    # Add subprograms here
    # Start of main program
    # Program generated by RoboDK v5.6.5 for UR10e on 02/02/2024 20:40:15
    # Using nominal kinematics.
    blend_radius_m = 0.001
    speed_ms = 1.000
    # set_reference(p[0.350000, -0.230000, -0.017000, 0.000000, 0.000000, 0.000000])
    set_tcp(p[0.000000, 0.000000, 0.252000, 0.000000, 0.000000, 0.000000])
    # Show Tool
    movej([-0.152532, -1.248081, -2.542110, -0.922198, 1.570796, 1.418264],accel_radss,speed_rads,0,blend_radius_m)
    movel([-0.152532, -1.248081, -2.542110, -0.922198, 1.570796, 1.418264],accel_mss,speed_ms,0,blend_radius_m)
    # Splitting Linear movement in 2 (instruction 7: MoveL 3)
    movel([-0.152532, -1.275419, -2.559682, -0.877288, 1.570796, 1.418264],accel_mss,speed_ms,0,blend_radius_m)
    movel([-0.152532, -1.305068, -2.576535, -0.830786, 1.570796, 1.418264],accel_mss,speed_ms,0,blend_radius_m)
    movel([-0.152532, -1.305068, -2.576535, -0.830786, 1.570796, 1.418264],accel_mss,speed_ms,0,blend_radius_m)
    speed_ms = 1.000
    movel([-0.152532, -1.305068, -2.576535, -0.830786, 1.570796, 1.418264],accel_mss,speed_ms,0,blend_radius_m)
    movel([-0.152532, -1.305068, -2.576535, -0.830786, 1.570796, 1.418264],accel_mss,speed_ms,0,blend_radius_m)
    movel([-0.152532, -1.305068, -2.576535, -0.830786, 1.570796, 1.418264],accel_mss,speed_ms,0,blend_radius_m)
    speed_ms = 0.005
    # Splitting Linear movement in 2 (instruction 14: MoveL 8)
    movel([-0.152532, -1.285041, -2.565382, -0.861966, 1.570796, 1.418264],accel_mss,speed_ms,0,blend_radius_m)
    movel([-0.152532, -1.266054, -2.553902, -0.892433, 1.570796, 1.418264],accel_mss,speed_ms,0,blend_radius_m)
    speed_ms = 1.000
    # Splitting Linear movement in 2 (instruction 16: MoveL 9)
    movel([-0.152532, -1.285041, -2.565382, -0.861966, 1.570796, 1.418264],accel_mss,speed_ms,0,blend_radius_m)
    movel([-0.152532, -1.305068, -2.576535, -0.830786, 1.570796, 1.418264],accel_mss,speed_ms,0,blend_radius_m)
    speed_ms = 0.040
    movel([-0.152532, -1.305068, -2.576535, -0.830786, 1.570796, 1.418264],accel_mss,speed_ms,0,blend_radius_m)
    speed_ms = 1.000
    movel([-0.152532, -1.305068, -2.576535, -0.830786, 1.570796, 1.418264],accel_mss,speed_ms,0,blend_radius_m)
    # Splitting Linear movement in 8 (instruction 21: MoveL 12)
    movel([-0.122948, -1.317915, -2.568481, -0.825992, 1.570796, 1.447849],accel_mss,speed_ms,0,blend_radius_m)
    movel([-0.094642, -1.331738, -2.559579, -0.821073, 1.570796, 1.476154],accel_mss,speed_ms,0,blend_radius_m)
    movel([-0.067601, -1.346424, -2.549844, -0.816120, 1.570796, 1.503196],accel_mss,speed_ms,0,blend_radius_m)
    movel([-0.041798, -1.361869, -2.539298, -0.811223, 1.570796, 1.528999],accel_mss,speed_ms,0,blend_radius_m)
    movel([-0.017201, -1.377969, -2.527959, -0.806462, 1.570796, 1.553595],accel_mss,speed_ms,0,blend_radius_m)
    movel([0.006227, -1.394629, -2.515848, -0.801912, 1.570796, 1.577023],accel_mss,speed_ms,0,blend_radius_m)
    movel([0.028528, -1.411761, -2.502989, -0.797639, 1.570796, 1.599324],accel_mss,speed_ms,0,blend_radius_m)
    movel([0.049747, -1.429285, -2.489403, -0.793702, 1.570796, 1.620543],accel_mss,speed_ms,0,blend_radius_m)
    speed_ms = 0.005
    # Splitting Linear movement in 2 (instruction 23: MoveL 13)
    movel([0.049747, -1.448539, -2.498917, -0.764933, 1.570796, 1.620543],accel_mss,speed_ms,0,blend_radius_m)
    movel([0.049747, -1.468584, -2.508071, -0.735733, 1.570796, 1.620543],accel_mss,speed_ms,0,blend_radius_m)
    speed_ms = 0.025
    movel([0.047987, -1.472694, -2.504618, -0.735077, 1.570796, 1.618783],accel_mss,speed_ms,0,blend_radius_m)
    movel([0.046994, -1.474744, -2.502886, -0.734759, 1.570796, 1.617791],accel_mss,speed_ms,0,blend_radius_m)
    movel([0.045905, -1.476777, -2.501162, -0.734450, 1.570796, 1.616702],accel_mss,speed_ms,0,blend_radius_m)
    movel([0.044706, -1.478782, -2.499455, -0.734152, 1.570796, 1.615502],accel_mss,speed_ms,0,blend_radius_m)
    movel([0.043381, -1.480749, -2.497774, -0.733866, 1.570796, 1.614178],accel_mss,speed_ms,0,blend_radius_m)
    movel([0.041915, -1.482668, -2.496128, -0.733593, 1.570796, 1.612712],accel_mss,speed_ms,0,blend_radius_m)
    movel([0.040291, -1.484527, -2.494529, -0.733333, 1.570796, 1.611088],accel_mss,speed_ms,0,blend_radius_m)
    movel([0.040888, -1.483683, -2.495255, -0.733450, 1.570796, 1.611684],accel_mss,speed_ms,0,blend_radius_m)
    movel([0.041419, -1.482572, -2.496211, -0.733606, 1.570796, 1.612216],accel_mss,speed_ms,0,blend_radius_m)
    movel([0.041720, -1.481480, -2.497148, -0.733761, 1.570796, 1.612517],accel_mss,speed_ms,0,blend_radius_m)
    movel([0.041730, -1.481035, -2.497529, -0.733825, 1.570796, 1.612526],accel_mss,speed_ms,0,blend_radius_m)
    movel([0.041619, -1.480703, -2.497813, -0.733873, 1.570796, 1.612415],accel_mss,speed_ms,0,blend_radius_m)
    movel([0.041364, -1.480515, -2.497974, -0.733900, 1.570796, 1.612160],accel_mss,speed_ms,0,blend_radius_m)
    movel([0.041013, -1.480523, -2.497967, -0.733899, 1.570796, 1.611810],accel_mss,speed_ms,0,blend_radius_m)
    movel([0.040586, -1.480703, -2.497813, -0.733873, 1.570796, 1.611382],accel_mss,speed_ms,0,blend_radius_m)
    movel([0.040090, -1.481034, -2.497530, -0.733825, 1.570796, 1.610886],accel_mss,speed_ms,0,blend_radius_m)
    movel([0.038959, -1.482046, -2.496663, -0.733681, 1.570796, 1.609755],accel_mss,speed_ms,0,blend_radius_m)
    movel([0.037732, -1.483368, -2.495527, -0.733494, 1.570796, 1.608528],accel_mss,speed_ms,0,blend_radius_m)
    movel([0.035425, -1.486199, -2.493085, -0.733105, 1.570796, 1.606222],accel_mss,speed_ms,0,blend_radius_m)
    movel([0.034030, -1.488028, -2.491501, -0.732860, 1.570796, 1.604827],accel_mss,speed_ms,0,blend_radius_m)
    movel([0.031932, -1.490562, -2.489297, -0.732529, 1.570796, 1.602728],accel_mss,speed_ms,0,blend_radius_m)
    movel([0.030757, -1.491738, -2.488272, -0.732379, 1.570796, 1.601553],accel_mss,speed_ms,0,blend_radius_m)
    movel([0.029446, -1.492789, -2.487353, -0.732247, 1.570796, 1.600242],accel_mss,speed_ms,0,blend_radius_m)
    movel([0.029713, -1.492441, -2.487658, -0.732291, 1.570796, 1.600509],accel_mss,speed_ms,0,blend_radius_m)
    movel([0.029890, -1.491885, -2.488143, -0.732361, 1.570796, 1.600686],accel_mss,speed_ms,0,blend_radius_m)
    movel([0.030008, -1.490434, -2.489409, -0.732546, 1.570796, 1.600805],accel_mss,speed_ms,0,blend_radius_m)
    movel([0.029868, -1.489016, -2.490643, -0.732730, 1.570796, 1.600664],accel_mss,speed_ms,0,blend_radius_m)
    movel([0.029718, -1.488499, -2.491093, -0.732798, 1.570796, 1.600514],accel_mss,speed_ms,0,blend_radius_m)
    movel([0.029529, -1.488209, -2.491344, -0.732836, 1.570796, 1.600325],accel_mss,speed_ms,0,blend_radius_m)
    movel([0.028992, -1.487953, -2.491566, -0.732870, 1.570796, 1.599789],accel_mss,speed_ms,0,blend_radius_m)
    movel([0.028458, -1.487944, -2.491574, -0.732871, 1.570796, 1.599254],accel_mss,speed_ms,0,blend_radius_m)
    movel([0.027927, -1.488133, -2.491410, -0.732846, 1.570796, 1.598724],accel_mss,speed_ms,0,blend_radius_m)
    movel([0.027405, -1.488475, -2.491113, -0.732801, 1.570796, 1.598201],accel_mss,speed_ms,0,blend_radius_m)
    movel([0.026411, -1.489409, -2.490302, -0.732678, 1.570796, 1.597207],accel_mss,speed_ms,0,blend_radius_m)
    movel([0.025512, -1.490359, -2.489474, -0.732555, 1.570796, 1.596308],accel_mss,speed_ms,0,blend_radius_m)
    movel([0.024026, -1.491761, -2.488251, -0.732376, 1.570796, 1.594822],accel_mss,speed_ms,0,blend_radius_m)
    movel([0.022503, -1.493004, -2.487165, -0.732220, 1.570796, 1.593300],accel_mss,speed_ms,0,blend_radius_m)
    movel([0.020851, -1.494060, -2.486240, -0.732089, 1.570796, 1.591648],accel_mss,speed_ms,0,blend_radius_m)
    movel([0.018986, -1.494894, -2.485508, -0.731987, 1.570796, 1.589782],accel_mss,speed_ms,0,blend_radius_m)
    movel([0.020018, -1.493786, -2.486480, -0.732123, 1.570796, 1.590814],accel_mss,speed_ms,0,blend_radius_m)
    movel([0.020844, -1.492612, -2.487508, -0.732269, 1.570796, 1.591641],accel_mss,speed_ms,0,blend_radius_m)
    movel([0.021097, -1.491990, -2.488052, -0.732347, 1.570796, 1.591893],accel_mss,speed_ms,0,blend_radius_m)
    movel([0.021184, -1.491389, -2.488577, -0.732423, 1.570796, 1.591981],accel_mss,speed_ms,0,blend_radius_m)
    movel([0.021086, -1.490859, -2.489039, -0.732491, 1.570796, 1.591883],accel_mss,speed_ms,0,blend_radius_m)
    movel([0.020770, -1.490458, -2.489389, -0.732543, 1.570796, 1.591566],accel_mss,speed_ms,0,blend_radius_m)
    movel([0.020101, -1.490219, -2.489596, -0.732573, 1.570796, 1.590897],accel_mss,speed_ms,0,blend_radius_m)
    movel([0.019264, -1.490254, -2.489566, -0.732569, 1.570796, 1.590061],accel_mss,speed_ms,0,blend_radius_m)
    movel([0.018340, -1.490477, -2.489372, -0.732540, 1.570796, 1.589137],accel_mss,speed_ms,0,blend_radius_m)
    movel([0.017414, -1.490797, -2.489093, -0.732499, 1.570796, 1.588211],accel_mss,speed_ms,0,blend_radius_m)
    speed_ms = 0.005
    movel([0.017414, -1.482861, -2.485566, -0.743963, 1.570796, 1.588211],accel_mss,speed_ms,0,blend_radius_m)
    speed_ms = 0.040
    movel([0.019926, -1.498929, -2.471530, -0.741930, 1.570796, 1.590722],accel_mss,speed_ms,0,blend_radius_m)
    speed_ms = 0.005
    movel([0.019926, -1.506737, -2.474994, -0.730658, 1.570796, 1.590722],accel_mss,speed_ms,0,blend_radius_m)
    speed_ms = 0.025
    movel([0.020345, -1.505703, -2.475921, -0.730765, 1.570796, 1.591141],accel_mss,speed_ms,0,blend_radius_m)
    movel([0.020900, -1.504675, -2.476841, -0.730873, 1.570796, 1.591696],accel_mss,speed_ms,0,blend_radius_m)
    movel([0.021577, -1.503669, -2.477739, -0.730981, 1.570796, 1.592373],accel_mss,speed_ms,0,blend_radius_m)
    movel([0.022366, -1.502696, -2.478607, -0.731086, 1.570796, 1.593163],accel_mss,speed_ms,0,blend_radius_m)
    movel([0.023256, -1.501770, -2.479431, -0.731188, 1.570796, 1.594052],accel_mss,speed_ms,0,blend_radius_m)
    movel([0.024233, -1.500906, -2.480198, -0.731285, 1.570796, 1.595030],accel_mss,speed_ms,0,blend_radius_m)
    movel([0.025286, -1.500119, -2.480897, -0.731373, 1.570796, 1.596082],accel_mss,speed_ms,0,blend_radius_m)
    movel([0.026405, -1.499419, -2.481517, -0.731453, 1.570796, 1.597201],accel_mss,speed_ms,0,blend_radius_m)
    movel([0.028138, -1.498558, -2.482279, -0.731552, 1.570796, 1.598935],accel_mss,speed_ms,0,blend_radius_m)
    movel([0.029837, -1.497950, -2.482816, -0.731623, 1.570796, 1.600634],accel_mss,speed_ms,0,blend_radius_m)
    movel([0.031496, -1.497576, -2.483146, -0.731667, 1.570796, 1.602293],accel_mss,speed_ms,0,blend_radius_m)
    movel([0.033106, -1.497418, -2.483285, -0.731685, 1.570796, 1.603903],accel_mss,speed_ms,0,blend_radius_m)
    movel([0.034662, -1.497458, -2.483250, -0.731681, 1.570796, 1.605458],accel_mss,speed_ms,0,blend_radius_m)
    movel([0.036159, -1.497677, -2.483057, -0.731655, 1.570796, 1.606956],accel_mss,speed_ms,0,blend_radius_m)
    movel([0.037589, -1.498057, -2.482722, -0.731610, 1.570796, 1.608386],accel_mss,speed_ms,0,blend_radius_m)
    movel([0.038948, -1.498578, -2.482261, -0.731550, 1.570796, 1.609744],accel_mss,speed_ms,0,blend_radius_m)
    movel([0.040230, -1.499221, -2.481692, -0.731476, 1.570796, 1.611026],accel_mss,speed_ms,0,blend_radius_m)
    movel([0.041430, -1.499967, -2.481031, -0.731391, 1.570796, 1.612227],accel_mss,speed_ms,0,blend_radius_m)
    movel([0.043569, -1.501692, -2.479500, -0.731197, 1.570796, 1.614365],accel_mss,speed_ms,0,blend_radius_m)
    movel([0.045328, -1.503594, -2.477806, -0.730989, 1.570796, 1.616124],accel_mss,speed_ms,0,blend_radius_m)
    movel([0.046669, -1.505525, -2.476080, -0.730784, 1.570796, 1.617465],accel_mss,speed_ms,0,blend_radius_m)
    movel([0.047792, -1.507678, -2.474150, -0.730562, 1.570796, 1.618588],accel_mss,speed_ms,0,blend_radius_m)
    movel([0.048705, -1.509943, -2.472110, -0.730336, 1.570796, 1.619501],accel_mss,speed_ms,0,blend_radius_m)
    movel([0.049431, -1.512301, -2.469978, -0.730110, 1.570796, 1.620227],accel_mss,speed_ms,0,blend_radius_m)
    movel([0.049991, -1.514735, -2.467768, -0.729886, 1.570796, 1.620788],accel_mss,speed_ms,0,blend_radius_m)
    movel([0.050411, -1.517225, -2.465497, -0.729667, 1.570796, 1.621207],accel_mss,speed_ms,0,blend_radius_m)
    movel([0.050713, -1.519754, -2.463181, -0.729454, 1.570796, 1.621510],accel_mss,speed_ms,0,blend_radius_m)
    movel([0.051058, -1.524854, -2.458479, -0.729056, 1.570796, 1.621854],accel_mss,speed_ms,0,blend_radius_m)
    movel([0.051259, -1.528417, -2.455169, -0.728803, 1.570796, 1.622055],accel_mss,speed_ms,0,blend_radius_m)
    movel([0.051521, -1.530125, -2.453575, -0.728689, 1.570796, 1.622318],accel_mss,speed_ms,0,blend_radius_m)
    movel([0.051999, -1.531735, -2.452069, -0.728586, 1.570796, 1.622795],accel_mss,speed_ms,0,blend_radius_m)
    movel([0.052951, -1.533693, -2.450230, -0.728465, 1.570796, 1.623747],accel_mss,speed_ms,0,blend_radius_m)
    movel([0.053905, -1.535658, -2.448380, -0.728351, 1.570796, 1.624701],accel_mss,speed_ms,0,blend_radius_m)
    movel([0.054234, -1.536676, -2.447418, -0.728294, 1.570796, 1.625030],accel_mss,speed_ms,0,blend_radius_m)
    movel([0.054384, -1.537737, -2.446415, -0.728237, 1.570796, 1.625180],accel_mss,speed_ms,0,blend_radius_m)
    movel([0.054296, -1.538850, -2.445360, -0.728179, 1.570796, 1.625093],accel_mss,speed_ms,0,blend_radius_m)
    movel([0.053915, -1.540032, -2.444238, -0.728119, 1.570796, 1.624711],accel_mss,speed_ms,0,blend_radius_m)
    movel([0.055176, -1.537118, -2.447000, -0.728270, 1.570796, 1.625972],accel_mss,speed_ms,0,blend_radius_m)
    movel([0.056268, -1.534210, -2.449744, -0.728435, 1.570796, 1.627064],accel_mss,speed_ms,0,blend_radius_m)
    movel([0.058142, -1.528367, -2.455216, -0.728806, 1.570796, 1.628938],accel_mss,speed_ms,0,blend_radius_m)
    movel([0.059066, -1.525102, -2.458249, -0.729038, 1.570796, 1.629862],accel_mss,speed_ms,0,blend_radius_m)
    movel([0.059888, -1.521837, -2.461266, -0.729287, 1.570796, 1.630684],accel_mss,speed_ms,0,blend_radius_m)
    movel([0.061298, -1.515293, -2.467260, -0.729836, 1.570796, 1.632094],accel_mss,speed_ms,0,blend_radius_m)
    movel([0.062426, -1.508876, -2.473071, -0.730441, 1.570796, 1.633222],accel_mss,speed_ms,0,blend_radius_m)
    movel([0.062809, -1.505673, -2.475948, -0.730768, 1.570796, 1.633605],accel_mss,speed_ms,0,blend_radius_m)
    movel([0.062991, -1.502530, -2.478754, -0.731105, 1.570796, 1.633787],accel_mss,speed_ms,0,blend_radius_m)
    movel([0.062929, -1.500110, -2.480905, -0.731374, 1.570796, 1.633725],accel_mss,speed_ms,0,blend_radius_m)
    movel([0.062735, -1.497714, -2.483025, -0.731651, 1.570796, 1.633532],accel_mss,speed_ms,0,blend_radius_m)
    movel([0.062551, -1.495294, -2.485157, -0.731939, 1.570796, 1.633347],accel_mss,speed_ms,0,blend_radius_m)
    movel([0.062514, -1.492802, -2.487341, -0.732245, 1.570796, 1.633310],accel_mss,speed_ms,0,blend_radius_m)
    movel([0.062598, -1.492115, -2.487942, -0.732331, 1.570796, 1.633394],accel_mss,speed_ms,0,blend_radius_m)
    movel([0.062833, -1.491405, -2.488563, -0.732421, 1.570796, 1.633629],accel_mss,speed_ms,0,blend_radius_m)
    movel([0.063253, -1.490783, -2.489105, -0.732501, 1.570796, 1.634049],accel_mss,speed_ms,0,blend_radius_m)
    movel([0.063548, -1.490538, -2.489318, -0.732532, 1.570796, 1.634344],accel_mss,speed_ms,0,blend_radius_m)
    movel([0.063906, -1.490355, -2.489478, -0.732556, 1.570796, 1.634702],accel_mss,speed_ms,0,blend_radius_m)
    movel([0.064424, -1.490247, -2.489573, -0.732570, 1.570796, 1.635220],accel_mss,speed_ms,0,blend_radius_m)
    movel([0.064916, -1.490252, -2.489568, -0.732569, 1.570796, 1.635712],accel_mss,speed_ms,0,blend_radius_m)
    movel([0.067510, -1.490558, -2.489301, -0.732530, 1.570796, 1.638306],accel_mss,speed_ms,0,blend_radius_m)
    movel([0.069847, -1.491127, -2.488805, -0.732457, 1.570796, 1.640644],accel_mss,speed_ms,0,blend_radius_m)
    movel([0.071947, -1.491931, -2.488103, -0.732355, 1.570796, 1.642743],accel_mss,speed_ms,0,blend_radius_m)
    movel([0.073826, -1.492954, -2.487208, -0.732226, 1.570796, 1.644622],accel_mss,speed_ms,0,blend_radius_m)
    movel([0.075502, -1.494170, -2.486143, -0.732076, 1.570796, 1.646298],accel_mss,speed_ms,0,blend_radius_m)
    movel([0.076994, -1.495556, -2.484926, -0.731907, 1.570796, 1.647790],accel_mss,speed_ms,0,blend_radius_m)
    movel([0.078319, -1.497090, -2.483575, -0.731724, 1.570796, 1.649115],accel_mss,speed_ms,0,blend_radius_m)
    movel([0.079494, -1.498753, -2.482106, -0.731530, 1.570796, 1.650290],accel_mss,speed_ms,0,blend_radius_m)
    movel([0.080539, -1.500520, -2.480541, -0.731328, 1.570796, 1.651335],accel_mss,speed_ms,0,blend_radius_m)
    movel([0.081473, -1.502370, -2.478897, -0.731122, 1.570796, 1.652270],accel_mss,speed_ms,0,blend_radius_m)
    movel([0.083080, -1.506232, -2.475447, -0.730710, 1.570796, 1.653876],accel_mss,speed_ms,0,blend_radius_m)
    movel([0.085758, -1.514035, -2.468404, -0.729950, 1.570796, 1.656554],accel_mss,speed_ms,0,blend_radius_m)
    movel([0.086253, -1.515217, -2.467329, -0.729843, 1.570796, 1.657050],accel_mss,speed_ms,0,blend_radius_m)
    movel([0.086622, -1.515721, -2.466870, -0.729798, 1.570796, 1.657418],accel_mss,speed_ms,0,blend_radius_m)
    movel([0.087122, -1.516115, -2.466511, -0.729763, 1.570796, 1.657919],accel_mss,speed_ms,0,blend_radius_m)
    movel([0.088103, -1.516424, -2.466228, -0.729736, 1.570796, 1.658899],accel_mss,speed_ms,0,blend_radius_m)
    movel([0.088627, -1.516441, -2.466213, -0.729735, 1.570796, 1.659423],accel_mss,speed_ms,0,blend_radius_m)
    movel([0.089168, -1.516374, -2.466274, -0.729741, 1.570796, 1.659965],accel_mss,speed_ms,0,blend_radius_m)
    movel([0.090276, -1.516027, -2.466591, -0.729771, 1.570796, 1.661072],accel_mss,speed_ms,0,blend_radius_m)
    movel([0.091387, -1.515445, -2.467122, -0.729823, 1.570796, 1.662183],accel_mss,speed_ms,0,blend_radius_m)
    movel([0.092457, -1.514694, -2.467805, -0.729890, 1.570796, 1.663254],accel_mss,speed_ms,0,blend_radius_m)
    movel([0.093445, -1.513838, -2.468584, -0.729968, 1.570796, 1.664242],accel_mss,speed_ms,0,blend_radius_m)
    movel([0.094311, -1.512937, -2.469401, -0.730051, 1.570796, 1.665107],accel_mss,speed_ms,0,blend_radius_m)
    movel([0.095004, -1.512057, -2.470199, -0.730133, 1.570796, 1.665800],accel_mss,speed_ms,0,blend_radius_m)
    movel([0.096042, -1.510510, -2.471598, -0.730281, 1.570796, 1.666838],accel_mss,speed_ms,0,blend_radius_m)
    movel([0.097003, -1.508932, -2.473021, -0.730436, 1.570796, 1.667799],accel_mss,speed_ms,0,blend_radius_m)
    movel([0.098688, -1.505713, -2.475912, -0.730764, 1.570796, 1.669484],accel_mss,speed_ms,0,blend_radius_m)
    movel([0.100061, -1.502456, -2.478820, -0.731113, 1.570796, 1.670857],accel_mss,speed_ms,0,blend_radius_m)
    movel([0.101119, -1.499219, -2.481694, -0.731476, 1.570796, 1.671915],accel_mss,speed_ms,0,blend_radius_m)
    movel([0.101462, -1.498003, -2.482769, -0.731617, 1.570796, 1.672258],accel_mss,speed_ms,0,blend_radius_m)
    movel([0.101921, -1.496793, -2.483837, -0.731759, 1.570796, 1.672717],accel_mss,speed_ms,0,blend_radius_m)
    movel([0.102246, -1.496209, -2.484351, -0.731829, 1.570796, 1.673043],accel_mss,speed_ms,0,blend_radius_m)
    movel([0.102663, -1.495646, -2.484847, -0.731896, 1.570796, 1.673459],accel_mss,speed_ms,0,blend_radius_m)
    movel([0.103191, -1.495113, -2.485315, -0.731961, 1.570796, 1.673987],accel_mss,speed_ms,0,blend_radius_m)
    movel([0.103850, -1.494618, -2.485750, -0.732021, 1.570796, 1.674647],accel_mss,speed_ms,0,blend_radius_m)
    movel([0.104844, -1.494159, -2.486153, -0.732077, 1.570796, 1.675640],accel_mss,speed_ms,0,blend_radius_m)
    movel([0.105852, -1.494002, -2.486291, -0.732096, 1.570796, 1.676648],accel_mss,speed_ms,0,blend_radius_m)
    movel([0.106800, -1.494096, -2.486208, -0.732085, 1.570796, 1.677597],accel_mss,speed_ms,0,blend_radius_m)
    movel([0.107623, -1.494391, -2.485949, -0.732049, 1.570796, 1.678419],accel_mss,speed_ms,0,blend_radius_m)
    movel([0.108793, -1.495109, -2.485319, -0.731961, 1.570796, 1.679590],accel_mss,speed_ms,0,blend_radius_m)
    movel([0.109841, -1.495969, -2.484562, -0.731857, 1.570796, 1.680638],accel_mss,speed_ms,0,blend_radius_m)
    movel([0.111647, -1.497907, -2.482854, -0.731628, 1.570796, 1.682444],accel_mss,speed_ms,0,blend_radius_m)
    movel([0.112379, -1.498899, -2.481977, -0.731513, 1.570796, 1.683175],accel_mss,speed_ms,0,blend_radius_m)
    movel([0.112973, -1.499942, -2.481054, -0.731393, 1.570796, 1.683770],accel_mss,speed_ms,0,blend_radius_m)
    movel([0.113440, -1.501029, -2.480089, -0.731271, 1.570796, 1.684237],accel_mss,speed_ms,0,blend_radius_m)
    movel([0.113785, -1.502160, -2.479084, -0.731145, 1.570796, 1.684581],accel_mss,speed_ms,0,blend_radius_m)
    movel([0.114013, -1.503328, -2.478044, -0.731018, 1.570796, 1.684810],accel_mss,speed_ms,0,blend_radius_m)
    movel([0.114151, -1.505768, -2.475863, -0.730758, 1.570796, 1.684947],accel_mss,speed_ms,0,blend_radius_m)
    movel([0.114072, -1.507032, -2.474729, -0.730628, 1.570796, 1.684869],accel_mss,speed_ms,0,blend_radius_m)
    movel([0.113660, -1.509630, -2.472392, -0.730367, 1.570796, 1.684456],accel_mss,speed_ms,0,blend_radius_m)
    movel([0.112946, -1.512298, -2.469980, -0.730110, 1.570796, 1.683743],accel_mss,speed_ms,0,blend_radius_m)
    movel([0.111984, -1.515015, -2.467513, -0.729861, 1.570796, 1.682780],accel_mss,speed_ms,0,blend_radius_m)
    movel([0.110827, -1.517747, -2.465020, -0.729622, 1.570796, 1.681624],accel_mss,speed_ms,0,blend_radius_m)
    movel([0.108876, -1.521723, -2.461371, -0.729296, 1.570796, 1.679673],accel_mss,speed_ms,0,blend_radius_m)
    movel([0.107771, -1.523695, -2.459551, -0.729143, 1.570796, 1.678567],accel_mss,speed_ms,0,blend_radius_m)
    movel([0.106563, -1.525642, -2.457749, -0.728999, 1.570796, 1.677359],accel_mss,speed_ms,0,blend_radius_m)
    movel([0.105242, -1.527548, -2.455978, -0.728863, 1.570796, 1.676038],accel_mss,speed_ms,0,blend_radius_m)
    movel([0.103799, -1.529403, -2.454250, -0.728737, 1.570796, 1.674595],accel_mss,speed_ms,0,blend_radius_m)
    movel([0.102219, -1.531196, -2.452573, -0.728620, 1.570796, 1.673015],accel_mss,speed_ms,0,blend_radius_m)
    movel([0.100495, -1.532914, -2.450963, -0.728513, 1.570796, 1.671291],accel_mss,speed_ms,0,blend_radius_m)
    movel([0.097886, -1.535185, -2.448826, -0.728378, 1.570796, 1.668682],accel_mss,speed_ms,0,blend_radius_m)
    movel([0.096431, -1.536300, -2.447774, -0.728315, 1.570796, 1.667227],accel_mss,speed_ms,0,blend_radius_m)
    movel([0.094906, -1.537331, -2.446799, -0.728259, 1.570796, 1.665702],accel_mss,speed_ms,0,blend_radius_m)
    movel([0.093336, -1.538226, -2.445951, -0.728211, 1.570796, 1.664133],accel_mss,speed_ms,0,blend_radius_m)
    movel([0.091746, -1.538933, -2.445281, -0.728174, 1.570796, 1.662542],accel_mss,speed_ms,0,blend_radius_m)
    movel([0.090156, -1.539398, -2.444841, -0.728151, 1.570796, 1.660953],accel_mss,speed_ms,0,blend_radius_m)
    movel([0.089370, -1.539524, -2.444720, -0.728144, 1.570796, 1.660167],accel_mss,speed_ms,0,blend_radius_m)
    movel([0.088595, -1.539569, -2.444678, -0.728142, 1.570796, 1.659391],accel_mss,speed_ms,0,blend_radius_m)
    movel([0.087751, -1.539517, -2.444727, -0.728145, 1.570796, 1.658547],accel_mss,speed_ms,0,blend_radius_m)
    movel([0.086976, -1.539361, -2.444875, -0.728153, 1.570796, 1.657772],accel_mss,speed_ms,0,blend_radius_m)
    movel([0.086265, -1.539111, -2.445113, -0.728165, 1.570796, 1.657062],accel_mss,speed_ms,0,blend_radius_m)
    movel([0.085615, -1.538774, -2.445432, -0.728183, 1.570796, 1.656412],accel_mss,speed_ms,0,blend_radius_m)
    movel([0.084479, -1.537886, -2.446274, -0.728229, 1.570796, 1.655275],accel_mss,speed_ms,0,blend_radius_m)
    movel([0.083539, -1.536771, -2.447329, -0.728289, 1.570796, 1.654335],accel_mss,speed_ms,0,blend_radius_m)
    movel([0.082764, -1.535510, -2.448519, -0.728360, 1.570796, 1.653560],accel_mss,speed_ms,0,blend_radius_m)
    movel([0.082122, -1.534181, -2.449771, -0.728436, 1.570796, 1.652919],accel_mss,speed_ms,0,blend_radius_m)
    movel([0.081123, -1.531634, -2.452163, -0.728592, 1.570796, 1.651920],accel_mss,speed_ms,0,blend_radius_m)
    movel([0.080674, -1.530439, -2.453281, -0.728668, 1.570796, 1.651470],accel_mss,speed_ms,0,blend_radius_m)
    movel([0.080087, -1.529336, -2.454312, -0.728741, 1.570796, 1.650883],accel_mss,speed_ms,0,blend_radius_m)
    movel([0.079683, -1.528878, -2.454739, -0.728772, 1.570796, 1.650479],accel_mss,speed_ms,0,blend_radius_m)
    movel([0.079173, -1.528514, -2.455079, -0.728796, 1.570796, 1.649970],accel_mss,speed_ms,0,blend_radius_m)
    movel([0.078537, -1.528269, -2.455307, -0.728813, 1.570796, 1.649333],accel_mss,speed_ms,0,blend_radius_m)
    movel([0.077749, -1.528165, -2.455404, -0.728820, 1.570796, 1.648545],accel_mss,speed_ms,0,blend_radius_m)
    movel([0.077921, -1.528219, -2.455353, -0.728817, 1.570796, 1.648717],accel_mss,speed_ms,0,blend_radius_m)
    movel([0.078022, -1.528366, -2.455217, -0.728807, 1.570796, 1.648818],accel_mss,speed_ms,0,blend_radius_m)
    movel([0.078024, -1.528912, -2.454707, -0.728769, 1.570796, 1.648821],accel_mss,speed_ms,0,blend_radius_m)
    movel([0.077786, -1.529757, -2.453919, -0.728713, 1.570796, 1.648582],accel_mss,speed_ms,0,blend_radius_m)
    movel([0.077343, -1.530853, -2.452894, -0.728642, 1.570796, 1.648140],accel_mss,speed_ms,0,blend_radius_m)
    movel([0.075981, -1.533606, -2.450312, -0.728471, 1.570796, 1.646777],accel_mss,speed_ms,0,blend_radius_m)
    movel([0.074205, -1.536791, -2.447310, -0.728288, 1.570796, 1.645001],accel_mss,speed_ms,0,blend_radius_m)
    movel([0.070469, -1.542969, -2.441439, -0.727980, 1.570796, 1.641265],accel_mss,speed_ms,0,blend_radius_m)
    movel([0.068192, -1.546458, -2.438097, -0.727834, 1.570796, 1.638988],accel_mss,speed_ms,0,blend_radius_m)
    movel([0.065488, -1.549998, -2.434686, -0.727705, 1.570796, 1.636284],accel_mss,speed_ms,0,blend_radius_m)
    movel([0.062729, -1.553454, -2.431336, -0.727599, 1.570796, 1.633525],accel_mss,speed_ms,0,blend_radius_m)
    movel([0.059905, -1.556864, -2.428013, -0.727513, 1.570796, 1.630702],accel_mss,speed_ms,0,blend_radius_m)
    movel([0.054252, -1.563384, -2.421604, -0.727401, 1.570796, 1.625048],accel_mss,speed_ms,0,blend_radius_m)
    movel([0.051363, -1.566407, -2.418610, -0.727372, 1.570796, 1.622159],accel_mss,speed_ms,0,blend_radius_m)
    movel([0.049836, -1.567837, -2.417189, -0.727363, 1.570796, 1.620632],accel_mss,speed_ms,0,blend_radius_m)
    movel([0.048242, -1.569190, -2.415840, -0.727358, 1.570796, 1.619039],accel_mss,speed_ms,0,blend_radius_m)
    movel([0.046566, -1.570450, -2.414583, -0.727356, 1.570796, 1.617363],accel_mss,speed_ms,0,blend_radius_m)
    movel([0.044802, -1.571600, -2.413433, -0.727357, 1.570796, 1.615598],accel_mss,speed_ms,0,blend_radius_m)
    movel([0.045149, -1.568689, -2.416340, -0.727360, 1.570796, 1.615946],accel_mss,speed_ms,0,blend_radius_m)
    movel([0.045119, -1.567858, -2.417168, -0.727363, 1.570796, 1.615916],accel_mss,speed_ms,0,blend_radius_m)
    movel([0.044947, -1.567542, -2.417483, -0.727365, 1.570796, 1.615743],accel_mss,speed_ms,0,blend_radius_m)
    movel([0.044607, -1.567377, -2.417647, -0.727366, 1.570796, 1.615403],accel_mss,speed_ms,0,blend_radius_m)
    movel([0.044234, -1.567394, -2.417629, -0.727366, 1.570796, 1.615030],accel_mss,speed_ms,0,blend_radius_m)
    movel([0.043838, -1.567527, -2.417497, -0.727365, 1.570796, 1.614635],accel_mss,speed_ms,0,blend_radius_m)
    movel([0.041962, -1.568497, -2.416532, -0.727361, 1.570796, 1.612759],accel_mss,speed_ms,0,blend_radius_m)
    movel([0.040849, -1.568905, -2.416124, -0.727359, 1.570796, 1.611646],accel_mss,speed_ms,0,blend_radius_m)
    movel([0.039732, -1.569172, -2.415858, -0.727358, 1.570796, 1.610528],accel_mss,speed_ms,0,blend_radius_m)
    movel([0.038640, -1.569290, -2.415741, -0.727358, 1.570796, 1.609436],accel_mss,speed_ms,0,blend_radius_m)
    movel([0.038311, -1.569242, -2.415789, -0.727358, 1.570796, 1.609108],accel_mss,speed_ms,0,blend_radius_m)
    movel([0.038215, -1.569055, -2.415975, -0.727359, 1.570796, 1.609011],accel_mss,speed_ms,0,blend_radius_m)
    movel([0.038508, -1.568213, -2.416814, -0.727362, 1.570796, 1.609304],accel_mss,speed_ms,0,blend_radius_m)
    movel([0.038473, -1.567947, -2.417080, -0.727363, 1.570796, 1.609269],accel_mss,speed_ms,0,blend_radius_m)
    movel([0.038291, -1.567758, -2.417267, -0.727364, 1.570796, 1.609087],accel_mss,speed_ms,0,blend_radius_m)
    movel([0.038010, -1.567656, -2.417369, -0.727364, 1.570796, 1.608806],accel_mss,speed_ms,0,blend_radius_m)
    movel([0.037675, -1.567648, -2.417377, -0.727364, 1.570796, 1.608472],accel_mss,speed_ms,0,blend_radius_m)
    movel([0.036971, -1.567857, -2.417169, -0.727363, 1.570796, 1.607768],accel_mss,speed_ms,0,blend_radius_m)
    movel([0.032034, -1.570539, -2.414494, -0.727356, 1.570796, 1.602831],accel_mss,speed_ms,0,blend_radius_m)
    movel([0.033488, -1.569504, -2.415528, -0.727358, 1.570796, 1.604284],accel_mss,speed_ms,0,blend_radius_m)
    movel([0.034915, -1.568368, -2.416660, -0.727361, 1.570796, 1.605712],accel_mss,speed_ms,0,blend_radius_m)
    movel([0.036304, -1.567153, -2.417869, -0.727367, 1.570796, 1.607100],accel_mss,speed_ms,0,blend_radius_m)
    movel([0.037649, -1.565876, -2.419138, -0.727376, 1.570796, 1.608445],accel_mss,speed_ms,0,blend_radius_m)
    movel([0.040174, -1.563204, -2.421782, -0.727403, 1.570796, 1.610970],accel_mss,speed_ms,0,blend_radius_m)
    movel([0.042420, -1.560504, -2.424443, -0.727442, 1.570796, 1.613216],accel_mss,speed_ms,0,blend_radius_m)
    movel([0.044692, -1.557524, -2.427367, -0.727498, 1.570796, 1.615489],accel_mss,speed_ms,0,blend_radius_m)
    movel([0.046838, -1.554469, -2.430349, -0.727571, 1.570796, 1.617635],accel_mss,speed_ms,0,blend_radius_m)
    movel([0.047827, -1.552916, -2.431859, -0.727614, 1.570796, 1.618623],accel_mss,speed_ms,0,blend_radius_m)
    movel([0.048742, -1.551347, -2.433381, -0.727661, 1.570796, 1.619539],accel_mss,speed_ms,0,blend_radius_m)
    movel([0.049567, -1.549765, -2.434911, -0.727713, 1.570796, 1.620363],accel_mss,speed_ms,0,blend_radius_m)
    movel([0.050288, -1.548168, -2.436452, -0.727769, 1.570796, 1.621084],accel_mss,speed_ms,0,blend_radius_m)
    movel([0.050654, -1.547170, -2.437413, -0.727806, 1.570796, 1.621451],accel_mss,speed_ms,0,blend_radius_m)
    movel([0.050929, -1.546167, -2.438377, -0.727845, 1.570796, 1.621725],accel_mss,speed_ms,0,blend_radius_m)
    movel([0.051225, -1.544162, -2.440299, -0.727928, 1.570796, 1.622021],accel_mss,speed_ms,0,blend_radius_m)
    movel([0.051211, -1.542184, -2.442189, -0.728016, 1.570796, 1.622007],accel_mss,speed_ms,0,blend_radius_m)
    movel([0.050919, -1.540264, -2.444018, -0.728108, 1.570796, 1.621716],accel_mss,speed_ms,0,blend_radius_m)
    movel([0.050389, -1.538428, -2.445760, -0.728201, 1.570796, 1.621186],accel_mss,speed_ms,0,blend_radius_m)
    movel([0.049659, -1.536708, -2.447388, -0.728293, 1.570796, 1.620455],accel_mss,speed_ms,0,blend_radius_m)
    movel([0.048760, -1.535134, -2.448874, -0.728381, 1.570796, 1.619557],accel_mss,speed_ms,0,blend_radius_m)
    movel([0.047734, -1.533734, -2.450192, -0.728463, 1.570796, 1.618531],accel_mss,speed_ms,0,blend_radius_m)
    movel([0.046969, -1.533087, -2.450800, -0.728502, 1.570796, 1.617766],accel_mss,speed_ms,0,blend_radius_m)
    movel([0.046036, -1.532733, -2.451133, -0.728524, 1.570796, 1.616832],accel_mss,speed_ms,0,blend_radius_m)
    movel([0.044989, -1.532658, -2.451202, -0.728528, 1.570796, 1.615785],accel_mss,speed_ms,0,blend_radius_m)
    movel([0.043886, -1.532851, -2.451022, -0.728516, 1.570796, 1.614683],accel_mss,speed_ms,0,blend_radius_m)
    movel([0.042779, -1.533292, -2.450607, -0.728490, 1.570796, 1.613575],accel_mss,speed_ms,0,blend_radius_m)
    movel([0.041722, -1.533971, -2.449969, -0.728449, 1.570796, 1.612519],accel_mss,speed_ms,0,blend_radius_m)
    movel([0.040776, -1.534867, -2.449125, -0.728396, 1.570796, 1.611572],accel_mss,speed_ms,0,blend_radius_m)
    movel([0.039990, -1.535966, -2.448089, -0.728334, 1.570796, 1.610787],accel_mss,speed_ms,0,blend_radius_m)
    movel([0.038953, -1.537691, -2.446459, -0.728239, 1.570796, 1.609749],accel_mss,speed_ms,0,blend_radius_m)
    movel([0.037826, -1.539382, -2.444855, -0.728152, 1.570796, 1.608622],accel_mss,speed_ms,0,blend_radius_m)
    movel([0.036599, -1.541021, -2.443297, -0.728071, 1.570796, 1.607395],accel_mss,speed_ms,0,blend_radius_m)
    movel([0.035257, -1.542593, -2.441799, -0.727997, 1.570796, 1.606053],accel_mss,speed_ms,0,blend_radius_m)
    movel([0.033791, -1.544077, -2.440380, -0.727932, 1.570796, 1.604587],accel_mss,speed_ms,0,blend_radius_m)
    movel([0.032187, -1.545460, -2.439055, -0.727874, 1.570796, 1.602984],accel_mss,speed_ms,0,blend_radius_m)
    movel([0.030433, -1.546725, -2.437841, -0.727823, 1.570796, 1.601229],accel_mss,speed_ms,0,blend_radius_m)
    movel([0.028519, -1.547854, -2.436755, -0.727781, 1.570796, 1.599315],accel_mss,speed_ms,0,blend_radius_m)
    movel([0.027475, -1.548332, -2.436294, -0.727763, 1.570796, 1.598272],accel_mss,speed_ms,0,blend_radius_m)
    movel([0.026412, -1.548698, -2.435941, -0.727750, 1.570796, 1.597208],accel_mss,speed_ms,0,blend_radius_m)
    movel([0.024268, -1.549225, -2.435433, -0.727731, 1.570796, 1.595065],accel_mss,speed_ms,0,blend_radius_m)
    movel([0.022596, -1.549491, -2.435176, -0.727722, 1.570796, 1.593392],accel_mss,speed_ms,0,blend_radius_m)
    movel([0.021010, -1.549563, -2.435106, -0.727720, 1.570796, 1.591806],accel_mss,speed_ms,0,blend_radius_m)
    movel([0.019511, -1.549457, -2.435209, -0.727723, 1.570796, 1.590308],accel_mss,speed_ms,0,blend_radius_m)
    movel([0.018095, -1.549187, -2.435470, -0.727733, 1.570796, 1.588891],accel_mss,speed_ms,0,blend_radius_m)
    movel([0.016758, -1.548771, -2.435871, -0.727747, 1.570796, 1.587554],accel_mss,speed_ms,0,blend_radius_m)
    movel([0.015496, -1.548222, -2.436399, -0.727767, 1.570796, 1.586293],accel_mss,speed_ms,0,blend_radius_m)
    movel([0.014313, -1.547556, -2.437041, -0.727792, 1.570796, 1.585109],accel_mss,speed_ms,0,blend_radius_m)
    movel([0.013202, -1.546790, -2.437779, -0.727821, 1.570796, 1.583999],accel_mss,speed_ms,0,blend_radius_m)
    movel([0.012162, -1.545938, -2.438597, -0.727854, 1.570796, 1.582959],accel_mss,speed_ms,0,blend_radius_m)
    movel([0.011193, -1.545012, -2.439485, -0.727892, 1.570796, 1.581989],accel_mss,speed_ms,0,blend_radius_m)
    movel([0.009457, -1.543013, -2.441397, -0.727978, 1.570796, 1.580253],accel_mss,speed_ms,0,blend_radius_m)
    movel([0.007979, -1.540912, -2.443401, -0.728076, 1.570796, 1.578775],accel_mss,speed_ms,0,blend_radius_m)
    movel([0.006747, -1.538836, -2.445373, -0.728179, 1.570796, 1.577544],accel_mss,speed_ms,0,blend_radius_m)
    movel([0.005914, -1.537189, -2.446933, -0.728266, 1.570796, 1.576710],accel_mss,speed_ms,0,blend_radius_m)
    movel([0.005168, -1.535434, -2.448591, -0.728364, 1.570796, 1.575964],accel_mss,speed_ms,0,blend_radius_m)
    movel([0.004519, -1.533579, -2.450338, -0.728472, 1.570796, 1.575315],accel_mss,speed_ms,0,blend_radius_m)
    movel([0.003986, -1.531636, -2.452161, -0.728592, 1.570796, 1.574783],accel_mss,speed_ms,0,blend_radius_m)
    movel([0.003580, -1.529616, -2.454051, -0.728722, 1.570796, 1.574376],accel_mss,speed_ms,0,blend_radius_m)
    movel([0.003317, -1.527529, -2.455996, -0.728864, 1.570796, 1.574114],accel_mss,speed_ms,0,blend_radius_m)
    movel([0.003214, -1.525386, -2.457986, -0.729017, 1.570796, 1.574010],accel_mss,speed_ms,0,blend_radius_m)
    movel([0.003284, -1.523198, -2.460010, -0.729181, 1.570796, 1.574081],accel_mss,speed_ms,0,blend_radius_m)
    movel([0.003542, -1.520975, -2.462059, -0.729355, 1.570796, 1.574338],accel_mss,speed_ms,0,blend_radius_m)
    movel([0.004003, -1.518731, -2.464119, -0.729539, 1.570796, 1.574800],accel_mss,speed_ms,0,blend_radius_m)
    movel([0.004683, -1.516473, -2.466184, -0.729732, 1.570796, 1.575479],accel_mss,speed_ms,0,blend_radius_m)
    movel([0.005599, -1.514215, -2.468241, -0.729933, 1.570796, 1.576396],accel_mss,speed_ms,0,blend_radius_m)
    movel([0.006765, -1.511969, -2.470278, -0.730141, 1.570796, 1.577561],accel_mss,speed_ms,0,blend_radius_m)
    movel([0.008199, -1.509745, -2.472288, -0.730356, 1.570796, 1.578995],accel_mss,speed_ms,0,blend_radius_m)
    movel([0.009913, -1.507560, -2.474255, -0.730574, 1.570796, 1.580709],accel_mss,speed_ms,0,blend_radius_m)
    movel([0.011923, -1.505424, -2.476171, -0.730794, 1.570796, 1.582720],accel_mss,speed_ms,0,blend_radius_m)
    movel([0.012797, -1.504654, -2.476860, -0.730876, 1.570796, 1.583593],accel_mss,speed_ms,0,blend_radius_m)
    movel([0.013277, -1.504331, -2.477148, -0.730910, 1.570796, 1.584073],accel_mss,speed_ms,0,blend_radius_m)
    movel([0.013789, -1.504089, -2.477364, -0.730936, 1.570796, 1.584585],accel_mss,speed_ms,0,blend_radius_m)
    movel([0.014561, -1.503942, -2.477496, -0.730952, 1.570796, 1.585357],accel_mss,speed_ms,0,blend_radius_m)
    movel([0.015250, -1.504040, -2.477408, -0.730941, 1.570796, 1.586046],accel_mss,speed_ms,0,blend_radius_m)
    movel([0.015830, -1.504330, -2.477149, -0.730910, 1.570796, 1.586626],accel_mss,speed_ms,0,blend_radius_m)
    movel([0.016270, -1.504757, -2.476767, -0.730865, 1.570796, 1.587067],accel_mss,speed_ms,0,blend_radius_m)
    movel([0.016900, -1.505930, -2.475718, -0.730741, 1.570796, 1.587696],accel_mss,speed_ms,0,blend_radius_m)
    movel([0.017252, -1.507271, -2.474515, -0.730603, 1.570796, 1.588049],accel_mss,speed_ms,0,blend_radius_m)
    movel([0.017654, -1.510076, -2.471990, -0.730323, 1.570796, 1.588450],accel_mss,speed_ms,0,blend_radius_m)
    movel([0.017877, -1.510551, -2.471561, -0.730277, 1.570796, 1.588673],accel_mss,speed_ms,0,blend_radius_m)
    movel([0.018117, -1.510629, -2.471491, -0.730270, 1.570796, 1.588914],accel_mss,speed_ms,0,blend_radius_m)
    movel([0.018485, -1.510569, -2.471544, -0.730275, 1.570796, 1.589281],accel_mss,speed_ms,0,blend_radius_m)
    movel([0.019067, -1.509442, -2.472562, -0.730385, 1.570796, 1.589864],accel_mss,speed_ms,0,blend_radius_m)
    movel([0.019568, -1.508284, -2.473604, -0.730501, 1.570796, 1.590365],accel_mss,speed_ms,0,blend_radius_m)
    movel([0.019982, -1.512436, -2.469855, -0.730098, 1.570796, 1.590778],accel_mss,speed_ms,0,blend_radius_m)
    movel([0.020558, -1.516505, -2.466155, -0.729729, 1.570796, 1.591354],accel_mss,speed_ms,0,blend_radius_m)
    movel([0.021295, -1.520487, -2.462508, -0.729394, 1.570796, 1.592091],accel_mss,speed_ms,0,blend_radius_m)
    movel([0.022191, -1.524383, -2.458915, -0.729091, 1.570796, 1.592987],accel_mss,speed_ms,0,blend_radius_m)
    movel([0.022649, -1.526045, -2.457375, -0.728969, 1.570796, 1.593445],accel_mss,speed_ms,0,blend_radius_m)
    movel([0.023296, -1.527701, -2.455836, -0.728852, 1.570796, 1.594092],accel_mss,speed_ms,0,blend_radius_m)
    movel([0.023724, -1.528467, -2.455122, -0.728800, 1.570796, 1.594520],accel_mss,speed_ms,0,blend_radius_m)
    movel([0.024238, -1.529159, -2.454478, -0.728753, 1.570796, 1.595035],accel_mss,speed_ms,0,blend_radius_m)
    movel([0.024855, -1.529751, -2.453924, -0.728713, 1.570796, 1.595651],accel_mss,speed_ms,0,blend_radius_m)
    movel([0.025587, -1.530219, -2.453487, -0.728683, 1.570796, 1.596384],accel_mss,speed_ms,0,blend_radius_m)
    movel([0.026170, -1.530452, -2.453270, -0.728668, 1.570796, 1.596966],accel_mss,speed_ms,0,blend_radius_m)
    movel([0.027457, -1.530642, -2.453092, -0.728655, 1.570796, 1.598253],accel_mss,speed_ms,0,blend_radius_m)
    movel([0.028149, -1.530613, -2.453119, -0.728657, 1.570796, 1.598945],accel_mss,speed_ms,0,blend_radius_m)
    movel([0.029599, -1.530339, -2.453375, -0.728675, 1.570796, 1.600395],accel_mss,speed_ms,0,blend_radius_m)
    movel([0.031098, -1.529820, -2.453860, -0.728709, 1.570796, 1.601894],accel_mss,speed_ms,0,blend_radius_m)
    movel([0.032596, -1.529109, -2.454524, -0.728756, 1.570796, 1.603392],accel_mss,speed_ms,0,blend_radius_m)
    movel([0.034042, -1.528253, -2.455322, -0.728814, 1.570796, 1.604839],accel_mss,speed_ms,0,blend_radius_m)
    movel([0.035389, -1.527306, -2.456203, -0.728880, 1.570796, 1.606186],accel_mss,speed_ms,0,blend_radius_m)
    movel([0.036582, -1.526318, -2.457121, -0.728950, 1.570796, 1.607378],accel_mss,speed_ms,0,blend_radius_m)
    speed_ms = 0.005
    movel([0.036582, -1.518669, -2.453733, -0.739987, 1.570796, 1.607378],accel_mss,speed_ms,0,blend_radius_m)
    speed_ms = 0.040
    movel([0.029707, -1.520999, -2.451592, -0.739798, 1.570796, 1.600503],accel_mss,speed_ms,0,blend_radius_m)
    speed_ms = 0.005
    movel([0.029707, -1.528629, -2.454972, -0.728789, 1.570796, 1.600503],accel_mss,speed_ms,0,blend_radius_m)
    speed_ms = 0.025
    movel([0.030662, -1.527790, -2.455753, -0.728846, 1.570796, 1.601458],accel_mss,speed_ms,0,blend_radius_m)
    movel([0.032483, -1.525887, -2.457521, -0.728981, 1.570796, 1.603279],accel_mss,speed_ms,0,blend_radius_m)
    movel([0.033332, -1.524844, -2.458488, -0.729057, 1.570796, 1.604128],accel_mss,speed_ms,0,blend_radius_m)
    movel([0.034867, -1.522630, -2.460534, -0.729225, 1.570796, 1.605663],accel_mss,speed_ms,0,blend_radius_m)
    movel([0.036139, -1.520315, -2.462665, -0.729408, 1.570796, 1.606935],accel_mss,speed_ms,0,blend_radius_m)
    movel([0.036655, -1.519150, -2.463735, -0.729504, 1.570796, 1.607451],accel_mss,speed_ms,0,blend_radius_m)
    movel([0.037080, -1.517990, -2.464798, -0.729601, 1.570796, 1.607876],accel_mss,speed_ms,0,blend_radius_m)
    movel([0.037625, -1.515742, -2.466851, -0.729796, 1.570796, 1.608421],accel_mss,speed_ms,0,blend_radius_m)
    movel([0.037730, -1.514673, -2.467824, -0.729892, 1.570796, 1.608527],accel_mss,speed_ms,0,blend_radius_m)
    movel([0.037711, -1.513660, -2.468745, -0.729984, 1.570796, 1.608507],accel_mss,speed_ms,0,blend_radius_m)
    movel([0.037562, -1.512711, -2.469606, -0.730072, 1.570796, 1.608358],accel_mss,speed_ms,0,blend_radius_m)
    movel([0.037272, -1.511838, -2.470397, -0.730154, 1.570796, 1.608069],accel_mss,speed_ms,0,blend_radius_m)
    movel([0.036758, -1.510843, -2.471297, -0.730249, 1.570796, 1.607554],accel_mss,speed_ms,0,blend_radius_m)
    movel([0.036113, -1.509942, -2.472111, -0.730336, 1.570796, 1.606909],accel_mss,speed_ms,0,blend_radius_m)
    movel([0.035329, -1.509166, -2.472810, -0.730413, 1.570796, 1.606125],accel_mss,speed_ms,0,blend_radius_m)
    movel([0.034399, -1.508552, -2.473363, -0.730474, 1.570796, 1.605195],accel_mss,speed_ms,0,blend_radius_m)
    movel([0.033317, -1.508132, -2.473741, -0.730516, 1.570796, 1.604113],accel_mss,speed_ms,0,blend_radius_m)
    movel([0.032079, -1.507942, -2.473912, -0.730535, 1.570796, 1.602875],accel_mss,speed_ms,0,blend_radius_m)
    movel([0.030678, -1.508015, -2.473846, -0.730528, 1.570796, 1.601475],accel_mss,speed_ms,0,blend_radius_m)
    movel([0.029111, -1.508381, -2.473517, -0.730491, 1.570796, 1.599907],accel_mss,speed_ms,0,blend_radius_m)
    movel([0.028034, -1.508807, -2.473134, -0.730448, 1.570796, 1.598830],accel_mss,speed_ms,0,blend_radius_m)
    movel([0.026989, -1.509378, -2.472620, -0.730392, 1.570796, 1.597785],accel_mss,speed_ms,0,blend_radius_m)
    movel([0.026011, -1.510066, -2.471999, -0.730324, 1.570796, 1.596808],accel_mss,speed_ms,0,blend_radius_m)
    movel([0.025131, -1.510848, -2.471292, -0.730248, 1.570796, 1.595927],accel_mss,speed_ms,0,blend_radius_m)
    movel([0.024378, -1.511699, -2.470523, -0.730167, 1.570796, 1.595174],accel_mss,speed_ms,0,blend_radius_m)
    movel([0.023782, -1.512594, -2.469713, -0.730083, 1.570796, 1.594578],accel_mss,speed_ms,0,blend_radius_m)
    movel([0.023377, -1.513506, -2.468884, -0.729998, 1.570796, 1.594173],accel_mss,speed_ms,0,blend_radius_m)
    movel([0.023187, -1.514415, -2.468059, -0.729915, 1.570796, 1.593984],accel_mss,speed_ms,0,blend_radius_m)
    speed_ms = 0.005
    movel([0.023187, -1.506669, -2.464625, -0.741095, 1.570796, 1.593984],accel_mss,speed_ms,0,blend_radius_m)
    speed_ms = 0.040
    # Splitting Linear movement in 2 (instruction 399: MoveL 378)
    movel([0.051290, -1.516388, -2.455821, -0.740180, 1.570796, 1.622087],accel_mss,speed_ms,0,blend_radius_m)
    movel([0.078430, -1.526900, -2.446130, -0.739359, 1.570796, 1.649227],accel_mss,speed_ms,0,blend_radius_m)
    speed_ms = 0.005
    movel([0.078430, -1.534483, -2.449487, -0.728419, 1.570796, 1.649227],accel_mss,speed_ms,0,blend_radius_m)
    speed_ms = 0.025
    movel([0.077845, -1.539171, -2.445055, -0.728162, 1.570796, 1.648641],accel_mss,speed_ms,0,blend_radius_m)
    movel([0.077355, -1.541529, -2.442814, -0.728047, 1.570796, 1.648151],accel_mss,speed_ms,0,blend_radius_m)
    movel([0.076991, -1.542730, -2.441668, -0.727991, 1.570796, 1.647787],accel_mss,speed_ms,0,blend_radius_m)
    movel([0.076521, -1.543950, -2.440502, -0.727937, 1.570796, 1.647317],accel_mss,speed_ms,0,blend_radius_m)
    movel([0.075883, -1.545241, -2.439265, -0.727883, 1.570796, 1.646679],accel_mss,speed_ms,0,blend_radius_m)
    movel([0.075474, -1.545865, -2.438667, -0.727857, 1.570796, 1.646270],accel_mss,speed_ms,0,blend_radius_m)
    movel([0.074975, -1.546457, -2.438098, -0.727834, 1.570796, 1.645772],accel_mss,speed_ms,0,blend_radius_m)
    movel([0.074917, -1.545380, -2.439132, -0.727877, 1.570796, 1.645713],accel_mss,speed_ms,0,blend_radius_m)
    movel([0.074651, -1.544385, -2.440086, -0.727919, 1.570796, 1.645447],accel_mss,speed_ms,0,blend_radius_m)
    movel([0.074441, -1.544113, -2.440346, -0.727930, 1.570796, 1.645237],accel_mss,speed_ms,0,blend_radius_m)
    movel([0.074235, -1.544095, -2.440363, -0.727931, 1.570796, 1.645031],accel_mss,speed_ms,0,blend_radius_m)
    movel([0.074002, -1.544166, -2.440295, -0.727928, 1.570796, 1.644799],accel_mss,speed_ms,0,blend_radius_m)
    movel([0.073546, -1.544468, -2.440006, -0.727915, 1.570796, 1.644342],accel_mss,speed_ms,0,blend_radius_m)
    movel([0.072920, -1.545089, -2.439411, -0.727889, 1.570796, 1.643716],accel_mss,speed_ms,0,blend_radius_m)
    movel([0.072434, -1.545739, -2.438788, -0.727862, 1.570796, 1.643230],accel_mss,speed_ms,0,blend_radius_m)
    movel([0.072061, -1.546408, -2.438145, -0.727836, 1.570796, 1.642857],accel_mss,speed_ms,0,blend_radius_m)
    movel([0.071777, -1.547091, -2.437489, -0.727809, 1.570796, 1.642573],accel_mss,speed_ms,0,blend_radius_m)
    movel([0.070981, -1.549850, -2.434829, -0.727710, 1.570796, 1.641778],accel_mss,speed_ms,0,blend_radius_m)
    movel([0.070413, -1.551470, -2.433262, -0.727657, 1.570796, 1.641209],accel_mss,speed_ms,0,blend_radius_m)
    movel([0.069717, -1.553085, -2.431695, -0.727609, 1.570796, 1.640513],accel_mss,speed_ms,0,blend_radius_m)
    movel([0.068858, -1.554681, -2.430142, -0.727566, 1.570796, 1.639655],accel_mss,speed_ms,0,blend_radius_m)
    movel([0.067805, -1.556238, -2.428624, -0.727527, 1.570796, 1.638601],accel_mss,speed_ms,0,blend_radius_m)
    movel([0.068063, -1.554979, -2.429852, -0.727558, 1.570796, 1.638860],accel_mss,speed_ms,0,blend_radius_m)
    movel([0.067978, -1.553800, -2.431000, -0.727589, 1.570796, 1.638774],accel_mss,speed_ms,0,blend_radius_m)
    movel([0.067880, -1.553531, -2.431261, -0.727597, 1.570796, 1.638676],accel_mss,speed_ms,0,blend_radius_m)
    movel([0.067664, -1.553353, -2.431434, -0.727602, 1.570796, 1.638460],accel_mss,speed_ms,0,blend_radius_m)
    movel([0.067395, -1.553343, -2.431444, -0.727602, 1.570796, 1.638191],accel_mss,speed_ms,0,blend_radius_m)
    movel([0.067096, -1.553445, -2.431345, -0.727599, 1.570796, 1.637893],accel_mss,speed_ms,0,blend_radius_m)
    movel([0.066527, -1.553838, -2.430963, -0.727588, 1.570796, 1.637323],accel_mss,speed_ms,0,blend_radius_m)
    movel([0.065929, -1.554444, -2.430373, -0.727572, 1.570796, 1.636725],accel_mss,speed_ms,0,blend_radius_m)
    movel([0.065425, -1.555097, -2.429737, -0.727555, 1.570796, 1.636222],accel_mss,speed_ms,0,blend_radius_m)
    movel([0.064630, -1.556488, -2.428379, -0.727521, 1.570796, 1.635426],accel_mss,speed_ms,0,blend_radius_m)
    movel([0.063348, -1.559296, -2.425630, -0.727463, 1.570796, 1.634145],accel_mss,speed_ms,0,blend_radius_m)
    movel([0.062488, -1.560840, -2.424112, -0.727436, 1.570796, 1.633284],accel_mss,speed_ms,0,blend_radius_m)
    movel([0.061504, -1.562357, -2.422618, -0.727414, 1.570796, 1.632300],accel_mss,speed_ms,0,blend_radius_m)
    movel([0.060367, -1.563818, -2.421175, -0.727396, 1.570796, 1.631163],accel_mss,speed_ms,0,blend_radius_m)
    movel([0.059049, -1.565195, -2.419812, -0.727382, 1.570796, 1.629845],accel_mss,speed_ms,0,blend_radius_m)
    movel([0.059292, -1.564503, -2.420497, -0.727388, 1.570796, 1.630088],accel_mss,speed_ms,0,blend_radius_m)
    movel([0.059487, -1.563157, -2.421829, -0.727403, 1.570796, 1.630284],accel_mss,speed_ms,0,blend_radius_m)
    movel([0.059436, -1.562520, -2.422457, -0.727412, 1.570796, 1.630232],accel_mss,speed_ms,0,blend_radius_m)
    movel([0.059334, -1.562256, -2.422718, -0.727415, 1.570796, 1.630130],accel_mss,speed_ms,0,blend_radius_m)
    movel([0.059075, -1.562157, -2.422815, -0.727416, 1.570796, 1.629871],accel_mss,speed_ms,0,blend_radius_m)
    movel([0.058716, -1.562339, -2.422636, -0.727414, 1.570796, 1.629513],accel_mss,speed_ms,0,blend_radius_m)
    movel([0.057925, -1.562984, -2.422000, -0.727405, 1.570796, 1.628722],accel_mss,speed_ms,0,blend_radius_m)
    movel([0.057246, -1.563664, -2.421327, -0.727397, 1.570796, 1.628042],accel_mss,speed_ms,0,blend_radius_m)
    movel([0.056090, -1.565100, -2.419907, -0.727382, 1.570796, 1.626886],accel_mss,speed_ms,0,blend_radius_m)
    movel([0.054983, -1.566564, -2.418454, -0.727371, 1.570796, 1.625780],accel_mss,speed_ms,0,blend_radius_m)
    movel([0.054365, -1.567285, -2.417738, -0.727366, 1.570796, 1.625161],accel_mss,speed_ms,0,blend_radius_m)
    movel([0.053658, -1.567985, -2.417041, -0.727363, 1.570796, 1.624454],accel_mss,speed_ms,0,blend_radius_m)
    movel([0.051800, -1.569572, -2.415460, -0.727357, 1.570796, 1.622596],accel_mss,speed_ms,0,blend_radius_m)
    movel([0.049863, -1.571079, -2.413954, -0.727356, 1.570796, 1.620660],accel_mss,speed_ms,0,blend_radius_m)
    movel([0.047871, -1.572512, -2.412518, -0.727359, 1.570796, 1.618667],accel_mss,speed_ms,0,blend_radius_m)
    movel([0.045837, -1.573884, -2.411141, -0.727364, 1.570796, 1.616634],accel_mss,speed_ms,0,blend_radius_m)
    speed_ms = 0.005
    movel([0.045837, -1.566622, -2.407929, -0.737838, 1.570796, 1.616634],accel_mss,speed_ms,0,blend_radius_m)
    speed_ms = 0.040
    movel([0.029341, -1.549189, -2.425003, -0.738197, 1.570796, 1.600137],accel_mss,speed_ms,0,blend_radius_m)
    speed_ms = 0.005
    movel([0.029341, -1.556592, -2.428278, -0.727519, 1.570796, 1.600137],accel_mss,speed_ms,0,blend_radius_m)
    speed_ms = 0.025
    movel([0.029967, -1.556056, -2.428801, -0.727531, 1.570796, 1.600763],accel_mss,speed_ms,0,blend_radius_m)
    movel([0.030522, -1.555448, -2.429395, -0.727546, 1.570796, 1.601318],accel_mss,speed_ms,0,blend_radius_m)
    movel([0.031512, -1.554098, -2.430710, -0.727581, 1.570796, 1.602308],accel_mss,speed_ms,0,blend_radius_m)
    movel([0.032486, -1.552713, -2.432056, -0.727620, 1.570796, 1.603282],accel_mss,speed_ms,0,blend_radius_m)
    movel([0.033024, -1.552059, -2.432690, -0.727639, 1.570796, 1.603820],accel_mss,speed_ms,0,blend_radius_m)
    movel([0.033625, -1.551460, -2.433271, -0.727658, 1.570796, 1.604422],accel_mss,speed_ms,0,blend_radius_m)
    movel([0.034109, -1.551081, -2.433639, -0.727670, 1.570796, 1.604905],accel_mss,speed_ms,0,blend_radius_m)
    movel([0.034514, -1.550857, -2.433855, -0.727677, 1.570796, 1.605310],accel_mss,speed_ms,0,blend_radius_m)
    movel([0.034846, -1.550772, -2.433938, -0.727680, 1.570796, 1.605642],accel_mss,speed_ms,0,blend_radius_m)
    movel([0.035114, -1.550807, -2.433904, -0.727678, 1.570796, 1.605910],accel_mss,speed_ms,0,blend_radius_m)
    movel([0.035476, -1.551181, -2.433541, -0.727666, 1.570796, 1.606273],accel_mss,speed_ms,0,blend_radius_m)
    movel([0.035654, -1.551846, -2.432897, -0.727646, 1.570796, 1.606451],accel_mss,speed_ms,0,blend_radius_m)
    movel([0.035652, -1.553528, -2.431265, -0.727597, 1.570796, 1.606449],accel_mss,speed_ms,0,blend_radius_m)
    movel([0.035520, -1.554807, -2.430019, -0.727562, 1.570796, 1.606317],accel_mss,speed_ms,0,blend_radius_m)
    movel([0.036607, -1.553451, -2.431340, -0.727599, 1.570796, 1.607403],accel_mss,speed_ms,0,blend_radius_m)
    movel([0.037417, -1.552109, -2.432642, -0.727638, 1.570796, 1.608213],accel_mss,speed_ms,0,blend_radius_m)
    movel([0.038022, -1.550775, -2.433935, -0.727679, 1.570796, 1.608818],accel_mss,speed_ms,0,blend_radius_m)
    movel([0.038487, -1.549443, -2.435222, -0.727724, 1.570796, 1.609283],accel_mss,speed_ms,0,blend_radius_m)
    movel([0.039732, -1.545392, -2.439121, -0.727876, 1.570796, 1.610528],accel_mss,speed_ms,0,blend_radius_m)
    movel([0.040325, -1.544001, -2.440453, -0.727935, 1.570796, 1.611121],accel_mss,speed_ms,0,blend_radius_m)
    movel([0.040666, -1.543456, -2.440974, -0.727959, 1.570796, 1.611462],accel_mss,speed_ms,0,blend_radius_m)
    movel([0.041027, -1.543133, -2.441283, -0.727973, 1.570796, 1.611823],accel_mss,speed_ms,0,blend_radius_m)
    movel([0.041393, -1.542997, -2.441413, -0.727979, 1.570796, 1.612189],accel_mss,speed_ms,0,blend_radius_m)
    movel([0.041747, -1.543018, -2.441393, -0.727978, 1.570796, 1.612544],accel_mss,speed_ms,0,blend_radius_m)
    movel([0.042077, -1.543160, -2.441257, -0.727972, 1.570796, 1.612873],accel_mss,speed_ms,0,blend_radius_m)
    movel([0.042363, -1.543391, -2.441036, -0.727962, 1.570796, 1.613159],accel_mss,speed_ms,0,blend_radius_m)
    movel([0.042751, -1.543986, -2.440468, -0.727936, 1.570796, 1.613547],accel_mss,speed_ms,0,blend_radius_m)
    movel([0.042858, -1.544696, -2.439788, -0.727905, 1.570796, 1.613655],accel_mss,speed_ms,0,blend_radius_m)
    movel([0.042815, -1.545644, -2.438879, -0.727866, 1.570796, 1.613612],accel_mss,speed_ms,0,blend_radius_m)
    movel([0.042602, -1.547416, -2.437176, -0.727797, 1.570796, 1.613398],accel_mss,speed_ms,0,blend_radius_m)
    movel([0.043636, -1.544669, -2.439814, -0.727907, 1.570796, 1.614432],accel_mss,speed_ms,0,blend_radius_m)
    movel([0.044012, -1.543300, -2.441124, -0.727966, 1.570796, 1.614808],accel_mss,speed_ms,0,blend_radius_m)
    movel([0.044476, -1.540592, -2.443706, -0.728092, 1.570796, 1.615272],accel_mss,speed_ms,0,blend_radius_m)
    movel([0.044559, -1.539266, -2.444965, -0.728157, 1.570796, 1.615356],accel_mss,speed_ms,0,blend_radius_m)
    movel([0.044427, -1.536697, -2.447399, -0.728293, 1.570796, 1.615223],accel_mss,speed_ms,0,blend_radius_m)
    speed_ms = 0.005
    movel([0.044427, -1.529132, -2.444050, -0.739207, 1.570796, 1.615223],accel_mss,speed_ms,0,blend_radius_m)
    speed_ms = 0.040
    movel([0.034396, -1.539639, -2.434152, -0.738598, 1.570796, 1.605192],accel_mss,speed_ms,0,blend_radius_m)
    speed_ms = 0.005
    movel([0.034396, -1.547119, -2.437462, -0.727808, 1.570796, 1.605192],accel_mss,speed_ms,0,blend_radius_m)
    speed_ms = 0.025
    movel([0.033124, -1.548649, -2.435989, -0.727752, 1.570796, 1.603921],accel_mss,speed_ms,0,blend_radius_m)
    movel([0.031967, -1.550220, -2.434471, -0.727698, 1.570796, 1.602764],accel_mss,speed_ms,0,blend_radius_m)
    movel([0.029723, -1.553380, -2.431408, -0.727601, 1.570796, 1.600519],accel_mss,speed_ms,0,blend_radius_m)
    movel([0.028483, -1.554925, -2.429905, -0.727559, 1.570796, 1.599279],accel_mss,speed_ms,0,blend_radius_m)
    movel([0.027098, -1.556390, -2.428475, -0.727524, 1.570796, 1.597895],accel_mss,speed_ms,0,blend_radius_m)
    movel([0.025552, -1.557703, -2.427192, -0.727495, 1.570796, 1.596348],accel_mss,speed_ms,0,blend_radius_m)
    movel([0.024714, -1.558279, -2.426628, -0.727483, 1.570796, 1.595510],accel_mss,speed_ms,0,blend_radius_m)
    movel([0.023830, -1.558789, -2.426128, -0.727473, 1.570796, 1.594627],accel_mss,speed_ms,0,blend_radius_m)
    movel([0.024473, -1.558300, -2.426607, -0.727482, 1.570796, 1.595270],accel_mss,speed_ms,0,blend_radius_m)
    movel([0.025137, -1.557542, -2.427349, -0.727498, 1.570796, 1.595934],accel_mss,speed_ms,0,blend_radius_m)
    movel([0.025747, -1.556626, -2.428245, -0.727518, 1.570796, 1.596543],accel_mss,speed_ms,0,blend_radius_m)
    movel([0.026215, -1.555667, -2.429182, -0.727541, 1.570796, 1.597012],accel_mss,speed_ms,0,blend_radius_m)
    movel([0.026464, -1.554775, -2.430050, -0.727563, 1.570796, 1.597260],accel_mss,speed_ms,0,blend_radius_m)
    movel([0.026478, -1.554394, -2.430422, -0.727573, 1.570796, 1.597275],accel_mss,speed_ms,0,blend_radius_m)
    movel([0.026408, -1.554072, -2.430735, -0.727582, 1.570796, 1.597204],accel_mss,speed_ms,0,blend_radius_m)
    movel([0.026242, -1.553823, -2.430977, -0.727589, 1.570796, 1.597038],accel_mss,speed_ms,0,blend_radius_m)
    movel([0.025967, -1.553666, -2.431130, -0.727593, 1.570796, 1.596764],accel_mss,speed_ms,0,blend_radius_m)
    movel([0.025578, -1.553610, -2.431184, -0.727594, 1.570796, 1.596374],accel_mss,speed_ms,0,blend_radius_m)
    movel([0.025059, -1.553673, -2.431123, -0.727593, 1.570796, 1.595856],accel_mss,speed_ms,0,blend_radius_m)
    movel([0.024231, -1.554003, -2.430802, -0.727584, 1.570796, 1.595027],accel_mss,speed_ms,0,blend_radius_m)
    movel([0.020833, -1.556030, -2.428827, -0.727532, 1.570796, 1.591629],accel_mss,speed_ms,0,blend_radius_m)
    movel([0.019373, -1.556765, -2.428109, -0.727515, 1.570796, 1.590169],accel_mss,speed_ms,0,blend_radius_m)
    movel([0.017870, -1.557410, -2.427478, -0.727501, 1.570796, 1.588666],accel_mss,speed_ms,0,blend_radius_m)
    movel([0.016371, -1.557921, -2.426978, -0.727490, 1.570796, 1.587168],accel_mss,speed_ms,0,blend_radius_m)
    movel([0.014924, -1.558247, -2.426658, -0.727483, 1.570796, 1.585720],accel_mss,speed_ms,0,blend_radius_m)
    movel([0.013571, -1.558343, -2.426564, -0.727481, 1.570796, 1.584368],accel_mss,speed_ms,0,blend_radius_m)
    movel([0.012362, -1.558158, -2.426746, -0.727485, 1.570796, 1.583159],accel_mss,speed_ms,0,blend_radius_m)
    movel([0.012749, -1.558163, -2.426741, -0.727485, 1.570796, 1.583545],accel_mss,speed_ms,0,blend_radius_m)
    movel([0.013255, -1.558014, -2.426887, -0.727488, 1.570796, 1.584051],accel_mss,speed_ms,0,blend_radius_m)
    movel([0.014465, -1.557405, -2.427483, -0.727501, 1.570796, 1.585262],accel_mss,speed_ms,0,blend_radius_m)
    movel([0.015650, -1.556628, -2.428243, -0.727518, 1.570796, 1.586446],accel_mss,speed_ms,0,blend_radius_m)
    movel([0.016463, -1.555984, -2.428872, -0.727533, 1.570796, 1.587259],accel_mss,speed_ms,0,blend_radius_m)
    movel([0.016937, -1.555461, -2.429382, -0.727546, 1.570796, 1.587734],accel_mss,speed_ms,0,blend_radius_m)
    movel([0.017112, -1.555085, -2.429748, -0.727555, 1.570796, 1.587908],accel_mss,speed_ms,0,blend_radius_m)
    movel([0.017034, -1.554834, -2.429993, -0.727562, 1.570796, 1.587830],accel_mss,speed_ms,0,blend_radius_m)
    movel([0.016759, -1.554686, -2.430138, -0.727566, 1.570796, 1.587555],accel_mss,speed_ms,0,blend_radius_m)
    movel([0.015833, -1.554607, -2.430214, -0.727568, 1.570796, 1.586629],accel_mss,speed_ms,0,blend_radius_m)
    movel([0.014762, -1.554673, -2.430150, -0.727566, 1.570796, 1.585558],accel_mss,speed_ms,0,blend_radius_m)
    movel([0.012326, -1.554819, -2.430008, -0.727562, 1.570796, 1.583122],accel_mss,speed_ms,0,blend_radius_m)
    movel([0.009899, -1.554777, -2.430049, -0.727563, 1.570796, 1.580695],accel_mss,speed_ms,0,blend_radius_m)
    movel([0.008753, -1.554631, -2.430191, -0.727567, 1.570796, 1.579550],accel_mss,speed_ms,0,blend_radius_m)
    movel([0.007687, -1.554372, -2.430443, -0.727574, 1.570796, 1.578484],accel_mss,speed_ms,0,blend_radius_m)
    movel([0.006727, -1.553977, -2.430827, -0.727584, 1.570796, 1.577523],accel_mss,speed_ms,0,blend_radius_m)
    movel([0.005899, -1.553426, -2.431364, -0.727600, 1.570796, 1.576696],accel_mss,speed_ms,0,blend_radius_m)
    movel([0.007352, -1.553330, -2.431457, -0.727602, 1.570796, 1.578149],accel_mss,speed_ms,0,blend_radius_m)
    movel([0.008148, -1.553123, -2.431658, -0.727608, 1.570796, 1.578944],accel_mss,speed_ms,0,blend_radius_m)
    movel([0.008500, -1.552950, -2.431826, -0.727613, 1.570796, 1.579296],accel_mss,speed_ms,0,blend_radius_m)
    movel([0.008800, -1.552716, -2.432053, -0.727620, 1.570796, 1.579597],accel_mss,speed_ms,0,blend_radius_m)
    movel([0.008923, -1.552515, -2.432248, -0.727626, 1.570796, 1.579719],accel_mss,speed_ms,0,blend_radius_m)
    movel([0.008905, -1.552303, -2.432454, -0.727632, 1.570796, 1.579701],accel_mss,speed_ms,0,blend_radius_m)
    movel([0.008524, -1.551863, -2.432881, -0.727645, 1.570796, 1.579320],accel_mss,speed_ms,0,blend_radius_m)
    movel([0.007787, -1.551416, -2.433314, -0.727659, 1.570796, 1.578583],accel_mss,speed_ms,0,blend_radius_m)
    movel([0.006830, -1.550983, -2.433734, -0.727673, 1.570796, 1.577626],accel_mss,speed_ms,0,blend_radius_m)
    movel([0.003478, -1.549785, -2.434892, -0.727712, 1.570796, 1.574275],accel_mss,speed_ms,0,blend_radius_m)
    movel([0.002266, -1.549172, -2.435484, -0.727733, 1.570796, 1.573062],accel_mss,speed_ms,0,blend_radius_m)
    movel([0.001172, -1.548431, -2.436199, -0.727760, 1.570796, 1.571968],accel_mss,speed_ms,0,blend_radius_m)
    movel([0.000270, -1.547536, -2.437061, -0.727792, 1.570796, 1.571066],accel_mss,speed_ms,0,blend_radius_m)
    movel([-0.000379, -1.546461, -2.438095, -0.727834, 1.570796, 1.570417],accel_mss,speed_ms,0,blend_radius_m)
    movel([0.000737, -1.547091, -2.437489, -0.727809, 1.570796, 1.571534],accel_mss,speed_ms,0,blend_radius_m)
    movel([0.001435, -1.547315, -2.437273, -0.727801, 1.570796, 1.572231],accel_mss,speed_ms,0,blend_radius_m)
    movel([0.002114, -1.547316, -2.437272, -0.727801, 1.570796, 1.572911],accel_mss,speed_ms,0,blend_radius_m)
    movel([0.002763, -1.547052, -2.437526, -0.727811, 1.570796, 1.573560],accel_mss,speed_ms,0,blend_radius_m)
    movel([0.003154, -1.546657, -2.437906, -0.727826, 1.570796, 1.573950],accel_mss,speed_ms,0,blend_radius_m)
    movel([0.003271, -1.546193, -2.438352, -0.727844, 1.570796, 1.574067],accel_mss,speed_ms,0,blend_radius_m)
    movel([0.003102, -1.545720, -2.438806, -0.727863, 1.570796, 1.573898],accel_mss,speed_ms,0,blend_radius_m)
    movel([0.001694, -1.543429, -2.441000, -0.727960, 1.570796, 1.572491],accel_mss,speed_ms,0,blend_radius_m)
    movel([0.000629, -1.541006, -2.443311, -0.728071, 1.570796, 1.571425],accel_mss,speed_ms,0,blend_radius_m)
    movel([0.000249, -1.539716, -2.444538, -0.728135, 1.570796, 1.571046],accel_mss,speed_ms,0,blend_radius_m)
    movel([-0.000017, -1.538359, -2.445826, -0.728204, 1.570796, 1.570780],accel_mss,speed_ms,0,blend_radius_m)
    movel([-0.000159, -1.536921, -2.447187, -0.728281, 1.570796, 1.570638],accel_mss,speed_ms,0,blend_radius_m)
    movel([-0.000167, -1.535393, -2.448630, -0.728366, 1.570796, 1.570629],accel_mss,speed_ms,0,blend_radius_m)
    speed_ms = 0.005
    movel([-0.000167, -1.527817, -2.445276, -0.739295, 1.570796, 1.570629],accel_mss,speed_ms,0,blend_radius_m)
    speed_ms = 0.040
    movel([-0.022466, -1.518241, -2.454125, -0.740023, 1.570796, 1.548330],accel_mss,speed_ms,0,blend_radius_m)
    speed_ms = 0.005
    movel([-0.022466, -1.525894, -2.457515, -0.728980, 1.570796, 1.548330],accel_mss,speed_ms,0,blend_radius_m)
    speed_ms = 0.025
    movel([-0.020597, -1.523608, -2.459632, -0.729150, 1.570796, 1.550199],accel_mss,speed_ms,0,blend_radius_m)
    movel([-0.018803, -1.521289, -2.461770, -0.729330, 1.570796, 1.551993],accel_mss,speed_ms,0,blend_radius_m)
    movel([-0.015402, -1.516544, -2.466119, -0.729726, 1.570796, 1.555394],accel_mss,speed_ms,0,blend_radius_m)
    movel([-0.012257, -1.511675, -2.470545, -0.730169, 1.570796, 1.558539],accel_mss,speed_ms,0,blend_radius_m)
    movel([-0.009374, -1.506698, -2.475029, -0.730662, 1.570796, 1.561423],accel_mss,speed_ms,0,blend_radius_m)
    movel([-0.006758, -1.501628, -2.479557, -0.731204, 1.570796, 1.564039],accel_mss,speed_ms,0,blend_radius_m)
    movel([-0.004417, -1.496483, -2.484110, -0.731796, 1.570796, 1.566379],accel_mss,speed_ms,0,blend_radius_m)
    movel([-0.002357, -1.491285, -2.488667, -0.732437, 1.570796, 1.568439],accel_mss,speed_ms,0,blend_radius_m)
    movel([-0.000586, -1.486048, -2.493215, -0.733125, 1.570796, 1.570210],accel_mss,speed_ms,0,blend_radius_m)
    movel([0.000887, -1.480798, -2.497732, -0.733859, 1.570796, 1.571683],accel_mss,speed_ms,0,blend_radius_m)
    movel([0.002055, -1.475554, -2.502200, -0.734635, 1.570796, 1.572851],accel_mss,speed_ms,0,blend_radius_m)
    movel([0.002907, -1.470339, -2.506601, -0.735450, 1.570796, 1.573704],accel_mss,speed_ms,0,blend_radius_m)
    movel([0.003433, -1.465176, -2.510915, -0.736298, 1.570796, 1.574229],accel_mss,speed_ms,0,blend_radius_m)
    movel([0.003629, -1.460086, -2.515128, -0.737175, 1.570796, 1.574425],accel_mss,speed_ms,0,blend_radius_m)
    movel([0.003478, -1.455098, -2.519218, -0.738073, 1.570796, 1.574274],accel_mss,speed_ms,0,blend_radius_m)
    movel([0.002975, -1.450238, -2.523165, -0.738986, 1.570796, 1.573771],accel_mss,speed_ms,0,blend_radius_m)
    movel([0.001663, -1.443176, -2.528837, -0.740376, 1.570796, 1.572460],accel_mss,speed_ms,0,blend_radius_m)
    movel([0.001633, -1.441931, -2.529829, -0.740629, 1.570796, 1.572429],accel_mss,speed_ms,0,blend_radius_m)
    movel([0.001847, -1.440618, -2.530872, -0.740898, 1.570796, 1.572643],accel_mss,speed_ms,0,blend_radius_m)
    movel([0.002491, -1.438763, -2.532343, -0.741284, 1.570796, 1.573287],accel_mss,speed_ms,0,blend_radius_m)
    movel([0.003293, -1.437317, -2.533484, -0.741587, 1.570796, 1.574089],accel_mss,speed_ms,0,blend_radius_m)
    movel([0.003745, -1.436740, -2.533940, -0.741710, 1.570796, 1.574542],accel_mss,speed_ms,0,blend_radius_m)
    movel([0.004739, -1.435848, -2.534641, -0.741899, 1.570796, 1.575536],accel_mss,speed_ms,0,blend_radius_m)
    movel([0.005272, -1.435530, -2.534892, -0.741967, 1.570796, 1.576068],accel_mss,speed_ms,0,blend_radius_m)
    movel([0.006401, -1.435122, -2.535212, -0.742055, 1.570796, 1.577198],accel_mss,speed_ms,0,blend_radius_m)
    movel([0.007590, -1.434991, -2.535315, -0.742083, 1.570796, 1.578387],accel_mss,speed_ms,0,blend_radius_m)
    movel([0.008814, -1.435103, -2.535227, -0.742059, 1.570796, 1.579611],accel_mss,speed_ms,0,blend_radius_m)
    movel([0.010051, -1.435426, -2.534974, -0.741990, 1.570796, 1.580848],accel_mss,speed_ms,0,blend_radius_m)
    movel([0.011275, -1.435920, -2.534585, -0.741884, 1.570796, 1.582071],accel_mss,speed_ms,0,blend_radius_m)
    movel([0.012464, -1.436554, -2.534086, -0.741749, 1.570796, 1.583260],accel_mss,speed_ms,0,blend_radius_m)
    movel([0.014637, -1.438088, -2.532876, -0.741425, 1.570796, 1.585434],accel_mss,speed_ms,0,blend_radius_m)
    movel([0.016390, -1.439747, -2.531563, -0.741079, 1.570796, 1.587186],accel_mss,speed_ms,0,blend_radius_m)
    movel([0.017549, -1.441238, -2.530380, -0.740771, 1.570796, 1.588345],accel_mss,speed_ms,0,blend_radius_m)
    movel([0.018583, -1.443176, -2.528837, -0.740376, 1.570796, 1.589380],accel_mss,speed_ms,0,blend_radius_m)
    movel([0.019434, -1.445226, -2.527199, -0.739965, 1.570796, 1.590230],accel_mss,speed_ms,0,blend_radius_m)
    movel([0.020761, -1.449528, -2.523739, -0.739122, 1.570796, 1.591558],accel_mss,speed_ms,0,blend_radius_m)
    movel([0.021881, -1.453903, -2.520192, -0.738294, 1.570796, 1.592678],accel_mss,speed_ms,0,blend_radius_m)
    movel([0.023134, -1.458118, -2.516746, -0.737525, 1.570796, 1.593931],accel_mss,speed_ms,0,blend_radius_m)
    movel([0.024538, -1.461727, -2.513775, -0.736888, 1.570796, 1.595335],accel_mss,speed_ms,0,blend_radius_m)
    movel([0.025445, -1.463393, -2.512395, -0.736601, 1.570796, 1.596242],accel_mss,speed_ms,0,blend_radius_m)
    movel([0.026600, -1.464881, -2.511160, -0.736348, 1.570796, 1.597396],accel_mss,speed_ms,0,blend_radius_m)
    movel([0.027285, -1.465459, -2.510679, -0.736250, 1.570796, 1.598081],accel_mss,speed_ms,0,blend_radius_m)
    movel([0.027711, -1.465654, -2.510517, -0.736218, 1.570796, 1.598507],accel_mss,speed_ms,0,blend_radius_m)
    movel([0.028210, -1.465744, -2.510442, -0.736203, 1.570796, 1.599006],accel_mss,speed_ms,0,blend_radius_m)
    movel([0.028929, -1.465671, -2.510503, -0.736215, 1.570796, 1.599725],accel_mss,speed_ms,0,blend_radius_m)
    movel([0.029678, -1.465424, -2.510708, -0.736256, 1.570796, 1.600475],accel_mss,speed_ms,0,blend_radius_m)
    movel([0.031166, -1.464617, -2.511380, -0.736392, 1.570796, 1.601962],accel_mss,speed_ms,0,blend_radius_m)
    movel([0.032779, -1.463512, -2.512297, -0.736580, 1.570796, 1.603576],accel_mss,speed_ms,0,blend_radius_m)
    movel([0.034310, -1.462320, -2.513284, -0.736785, 1.570796, 1.605106],accel_mss,speed_ms,0,blend_radius_m)
    movel([0.037186, -1.459741, -2.515412, -0.737236, 1.570796, 1.607982],accel_mss,speed_ms,0,blend_radius_m)
    movel([0.042702, -1.454304, -2.519865, -0.738220, 1.570796, 1.613498],accel_mss,speed_ms,0,blend_radius_m)
    movel([0.045403, -1.451829, -2.521877, -0.738683, 1.570796, 1.616199],accel_mss,speed_ms,0,blend_radius_m)
    movel([0.046992, -1.450531, -2.522928, -0.738930, 1.570796, 1.617788],accel_mss,speed_ms,0,blend_radius_m)
    movel([0.048604, -1.449412, -2.523833, -0.739144, 1.570796, 1.619400],accel_mss,speed_ms,0,blend_radius_m)
    movel([0.049387, -1.448969, -2.524190, -0.739230, 1.570796, 1.620183],accel_mss,speed_ms,0,blend_radius_m)
    movel([0.050139, -1.448633, -2.524461, -0.739295, 1.570796, 1.620936],accel_mss,speed_ms,0,blend_radius_m)
    movel([0.050846, -1.448423, -2.524631, -0.739336, 1.570796, 1.621642],accel_mss,speed_ms,0,blend_radius_m)
    movel([0.051495, -1.448361, -2.524681, -0.739348, 1.570796, 1.622291],accel_mss,speed_ms,0,blend_radius_m)
    movel([0.052072, -1.448464, -2.524597, -0.739328, 1.570796, 1.622869],accel_mss,speed_ms,0,blend_radius_m)
    movel([0.052567, -1.448754, -2.524364, -0.739271, 1.570796, 1.623363],accel_mss,speed_ms,0,blend_radius_m)
    movel([0.052966, -1.449251, -2.523962, -0.739175, 1.570796, 1.623763],accel_mss,speed_ms,0,blend_radius_m)
    movel([0.053255, -1.449976, -2.523377, -0.739036, 1.570796, 1.624051],accel_mss,speed_ms,0,blend_radius_m)
    movel([0.053543, -1.451361, -2.522257, -0.738772, 1.570796, 1.624340],accel_mss,speed_ms,0,blend_radius_m)
    movel([0.053666, -1.452775, -2.521109, -0.738505, 1.570796, 1.624462],accel_mss,speed_ms,0,blend_radius_m)
    movel([0.053632, -1.454212, -2.519940, -0.738237, 1.570796, 1.624429],accel_mss,speed_ms,0,blend_radius_m)
    movel([0.053453, -1.455671, -2.518750, -0.737968, 1.570796, 1.624249],accel_mss,speed_ms,0,blend_radius_m)
    movel([0.053133, -1.457143, -2.517546, -0.737700, 1.570796, 1.623929],accel_mss,speed_ms,0,blend_radius_m)
    movel([0.052683, -1.458624, -2.516331, -0.737434, 1.570796, 1.623479],accel_mss,speed_ms,0,blend_radius_m)
    movel([0.052110, -1.460111, -2.515108, -0.737171, 1.570796, 1.622906],accel_mss,speed_ms,0,blend_radius_m)
    movel([0.051424, -1.461599, -2.513880, -0.736910, 1.570796, 1.622220],accel_mss,speed_ms,0,blend_radius_m)
    movel([0.049747, -1.464556, -2.511430, -0.736403, 1.570796, 1.620543],accel_mss,speed_ms,0,blend_radius_m)
    movel([0.047714, -1.467466, -2.509006, -0.735917, 1.570796, 1.618510],accel_mss,speed_ms,0,blend_radius_m)
    movel([0.045389, -1.470294, -2.506638, -0.735457, 1.570796, 1.616185],accel_mss,speed_ms,0,blend_radius_m)
    movel([0.042838, -1.473006, -2.504355, -0.735028, 1.570796, 1.613634],accel_mss,speed_ms,0,blend_radius_m)
    movel([0.036899, -1.478881, -2.499370, -0.734138, 1.570796, 1.607695],accel_mss,speed_ms,0,blend_radius_m)
    movel([0.033733, -1.481692, -2.496966, -0.733731, 1.570796, 1.604529],accel_mss,speed_ms,0,blend_radius_m)
    movel([0.032106, -1.482978, -2.495862, -0.733549, 1.570796, 1.602902],accel_mss,speed_ms,0,blend_radius_m)
    movel([0.030449, -1.484152, -2.494851, -0.733385, 1.570796, 1.601246],accel_mss,speed_ms,0,blend_radius_m)
    movel([0.029367, -1.484827, -2.494270, -0.733292, 1.570796, 1.600163],accel_mss,speed_ms,0,blend_radius_m)
    movel([0.028277, -1.485408, -2.493769, -0.733212, 1.570796, 1.599074],accel_mss,speed_ms,0,blend_radius_m)
    movel([0.027188, -1.485882, -2.493359, -0.733148, 1.570796, 1.597984],accel_mss,speed_ms,0,blend_radius_m)
    movel([0.026108, -1.486237, -2.493053, -0.733100, 1.570796, 1.596904],accel_mss,speed_ms,0,blend_radius_m)
    movel([0.025048, -1.486460, -2.492860, -0.733070, 1.570796, 1.595844],accel_mss,speed_ms,0,blend_radius_m)
    movel([0.024014, -1.486539, -2.492791, -0.733059, 1.570796, 1.594811],accel_mss,speed_ms,0,blend_radius_m)
    movel([0.023018, -1.486457, -2.492862, -0.733070, 1.570796, 1.593814],accel_mss,speed_ms,0,blend_radius_m)
    movel([0.022065, -1.486202, -2.493082, -0.733104, 1.570796, 1.592861],accel_mss,speed_ms,0,blend_radius_m)
    movel([0.021200, -1.485770, -2.493456, -0.733163, 1.570796, 1.591996],accel_mss,speed_ms,0,blend_radius_m)
    movel([0.020477, -1.485214, -2.493936, -0.733239, 1.570796, 1.591274],accel_mss,speed_ms,0,blend_radius_m)
    movel([0.018046, -1.482555, -2.496225, -0.733609, 1.570796, 1.588843],accel_mss,speed_ms,0,blend_radius_m)
    movel([0.017307, -1.481986, -2.496714, -0.733689, 1.570796, 1.588104],accel_mss,speed_ms,0,blend_radius_m)
    movel([0.016416, -1.481539, -2.497097, -0.733753, 1.570796, 1.587212],accel_mss,speed_ms,0,blend_radius_m)
    movel([0.016011, -1.481473, -2.497154, -0.733762, 1.570796, 1.586808],accel_mss,speed_ms,0,blend_radius_m)
    movel([0.015826, -1.481649, -2.497003, -0.733737, 1.570796, 1.586622],accel_mss,speed_ms,0,blend_radius_m)
    movel([0.015586, -1.482106, -2.496611, -0.733672, 1.570796, 1.586383],accel_mss,speed_ms,0,blend_radius_m)
    movel([0.014967, -1.483715, -2.495228, -0.733446, 1.570796, 1.585763],accel_mss,speed_ms,0,blend_radius_m)
    movel([0.013426, -1.488626, -2.490982, -0.732781, 1.570796, 1.584223],accel_mss,speed_ms,0,blend_radius_m)
    movel([0.011008, -1.496849, -2.483788, -0.731753, 1.570796, 1.581805],accel_mss,speed_ms,0,blend_radius_m)
    movel([0.009222, -1.501167, -2.479967, -0.731255, 1.570796, 1.580018],accel_mss,speed_ms,0,blend_radius_m)
    movel([0.007219, -1.505451, -2.476146, -0.730791, 1.570796, 1.578016],accel_mss,speed_ms,0,blend_radius_m)
    movel([0.005025, -1.509696, -2.472332, -0.730360, 1.570796, 1.575822],accel_mss,speed_ms,0,blend_radius_m)
    movel([0.002672, -1.513892, -2.468534, -0.729963, 1.570796, 1.573469],accel_mss,speed_ms,0,blend_radius_m)
    movel([-0.000478, -1.519211, -2.463679, -0.729499, 1.570796, 1.570319],accel_mss,speed_ms,0,blend_radius_m)
    movel([-0.003754, -1.524489, -2.458816, -0.729083, 1.570796, 1.567042],accel_mss,speed_ms,0,blend_radius_m)
    movel([-0.007182, -1.529699, -2.453973, -0.728717, 1.570796, 1.563614],accel_mss,speed_ms,0,blend_radius_m)
    movel([-0.010795, -1.534808, -2.449181, -0.728400, 1.570796, 1.560002],accel_mss,speed_ms,0,blend_radius_m)
    movel([-0.014617, -1.539786, -2.444472, -0.728131, 1.570796, 1.556179],accel_mss,speed_ms,0,blend_radius_m)
    movel([-0.016614, -1.542217, -2.442157, -0.728015, 1.570796, 1.554182],accel_mss,speed_ms,0,blend_radius_m)
    movel([-0.018676, -1.544606, -2.439874, -0.727909, 1.570796, 1.552120],accel_mss,speed_ms,0,blend_radius_m)
    movel([-0.020806, -1.546949, -2.437625, -0.727815, 1.570796, 1.549991],accel_mss,speed_ms,0,blend_radius_m)
    movel([-0.023005, -1.549240, -2.435418, -0.727731, 1.570796, 1.547792],accel_mss,speed_ms,0,blend_radius_m)
    movel([-0.025277, -1.551481, -2.433251, -0.727657, 1.570796, 1.545519],accel_mss,speed_ms,0,blend_radius_m)
    movel([-0.027630, -1.553663, -2.431133, -0.727593, 1.570796, 1.543167],accel_mss,speed_ms,0,blend_radius_m)
    movel([-0.030515, -1.556180, -2.428680, -0.727529, 1.570796, 1.540281],accel_mss,speed_ms,0,blend_radius_m)
    movel([-0.032020, -1.557367, -2.427521, -0.727502, 1.570796, 1.538776],accel_mss,speed_ms,0,blend_radius_m)
    movel([-0.034729, -1.559211, -2.425714, -0.727465, 1.570796, 1.536067],accel_mss,speed_ms,0,blend_radius_m)
    movel([-0.036131, -1.560015, -2.424924, -0.727450, 1.570796, 1.534665],accel_mss,speed_ms,0,blend_radius_m)
    movel([-0.037535, -1.560590, -2.424358, -0.727440, 1.570796, 1.533261],accel_mss,speed_ms,0,blend_radius_m)
    movel([-0.038157, -1.560699, -2.424252, -0.727438, 1.570796, 1.532640],accel_mss,speed_ms,0,blend_radius_m)
    movel([-0.038686, -1.560641, -2.424308, -0.727439, 1.570796, 1.532111],accel_mss,speed_ms,0,blend_radius_m)
    movel([-0.038269, -1.559366, -2.425562, -0.727462, 1.570796, 1.532527],accel_mss,speed_ms,0,blend_radius_m)
    movel([-0.038057, -1.558114, -2.426789, -0.727486, 1.570796, 1.532739],accel_mss,speed_ms,0,blend_radius_m)
    movel([-0.038080, -1.557546, -2.427345, -0.727498, 1.570796, 1.532717],accel_mss,speed_ms,0,blend_radius_m)
    movel([-0.038217, -1.557042, -2.427838, -0.727509, 1.570796, 1.532579],accel_mss,speed_ms,0,blend_radius_m)
    movel([-0.038489, -1.556621, -2.428249, -0.727518, 1.570796, 1.532307],accel_mss,speed_ms,0,blend_radius_m)
    movel([-0.038922, -1.556307, -2.428557, -0.727526, 1.570796, 1.531874],accel_mss,speed_ms,0,blend_radius_m)
    movel([-0.040266, -1.555847, -2.429006, -0.727536, 1.570796, 1.530530],accel_mss,speed_ms,0,blend_radius_m)
    movel([-0.040634, -1.555571, -2.429275, -0.727543, 1.570796, 1.530162],accel_mss,speed_ms,0,blend_radius_m)
    movel([-0.040882, -1.555212, -2.429625, -0.727552, 1.570796, 1.529914],accel_mss,speed_ms,0,blend_radius_m)
    movel([-0.041069, -1.554306, -2.430507, -0.727576, 1.570796, 1.529727],accel_mss,speed_ms,0,blend_radius_m)
    movel([-0.040955, -1.553246, -2.431538, -0.727605, 1.570796, 1.529841],accel_mss,speed_ms,0,blend_radius_m)
    movel([-0.040664, -1.552156, -2.432596, -0.727636, 1.570796, 1.530133],accel_mss,speed_ms,0,blend_radius_m)
    movel([-0.039553, -1.548866, -2.435779, -0.727744, 1.570796, 1.531243],accel_mss,speed_ms,0,blend_radius_m)
    movel([-0.038218, -1.545533, -2.438985, -0.727871, 1.570796, 1.532578],accel_mss,speed_ms,0,blend_radius_m)
    movel([-0.037429, -1.543870, -2.440578, -0.727941, 1.570796, 1.533368],accel_mss,speed_ms,0,blend_radius_m)
    movel([-0.036541, -1.542216, -2.442158, -0.728015, 1.570796, 1.534255],accel_mss,speed_ms,0,blend_radius_m)
    movel([-0.035539, -1.540583, -2.443714, -0.728092, 1.570796, 1.535257],accel_mss,speed_ms,0,blend_radius_m)
    movel([-0.034409, -1.538975, -2.445242, -0.728172, 1.570796, 1.536388],accel_mss,speed_ms,0,blend_radius_m)
    movel([-0.033134, -1.537476, -2.446662, -0.728251, 1.570796, 1.537662],accel_mss,speed_ms,0,blend_radius_m)
    movel([-0.028906, -1.533326, -2.450576, -0.728488, 1.570796, 1.541890],accel_mss,speed_ms,0,blend_radius_m)
    movel([-0.025637, -1.529653, -2.454016, -0.728720, 1.570796, 1.545159],accel_mss,speed_ms,0,blend_radius_m)
    movel([-0.022466, -1.525894, -2.457515, -0.728980, 1.570796, 1.548330],accel_mss,speed_ms,0,blend_radius_m)
    movel([-0.021068, -1.524181, -2.459101, -0.729106, 1.570796, 1.549729],accel_mss,speed_ms,0,blend_radius_m)
    speed_ms = 0.005
    movel([-0.021068, -1.516515, -2.455705, -0.740169, 1.570796, 1.549729],accel_mss,speed_ms,0,blend_radius_m)
    speed_ms = 0.040
    movel([-0.050485, -1.547182, -2.426938, -0.738269, 1.570796, 1.520312],accel_mss,speed_ms,0,blend_radius_m)
    speed_ms = 0.005
    movel([-0.050485, -1.554601, -2.430220, -0.727568, 1.570796, 1.520312],accel_mss,speed_ms,0,blend_radius_m)
    speed_ms = 0.025
    movel([-0.048077, -1.556856, -2.428020, -0.727513, 1.570796, 1.522719],accel_mss,speed_ms,0,blend_radius_m)
    movel([-0.046893, -1.558135, -2.426768, -0.727486, 1.570796, 1.523903],accel_mss,speed_ms,0,blend_radius_m)
    movel([-0.045817, -1.559516, -2.425414, -0.727459, 1.570796, 1.524979],accel_mss,speed_ms,0,blend_radius_m)
    movel([-0.044913, -1.560988, -2.423967, -0.727434, 1.570796, 1.525883],accel_mss,speed_ms,0,blend_radius_m)
    movel([-0.044250, -1.562548, -2.422429, -0.727411, 1.570796, 1.526546],accel_mss,speed_ms,0,blend_radius_m)
    movel([-0.043895, -1.564194, -2.420804, -0.727391, 1.570796, 1.526901],accel_mss,speed_ms,0,blend_radius_m)
    movel([-0.043854, -1.565048, -2.419958, -0.727383, 1.570796, 1.526942],accel_mss,speed_ms,0,blend_radius_m)
    movel([-0.043915, -1.565919, -2.419095, -0.727375, 1.570796, 1.526881],accel_mss,speed_ms,0,blend_radius_m)
    movel([-0.044514, -1.565604, -2.419407, -0.727378, 1.570796, 1.526282],accel_mss,speed_ms,0,blend_radius_m)
    movel([-0.044896, -1.565193, -2.419815, -0.727382, 1.570796, 1.525901],accel_mss,speed_ms,0,blend_radius_m)
    movel([-0.045696, -1.564234, -2.420764, -0.727391, 1.570796, 1.525100],accel_mss,speed_ms,0,blend_radius_m)
    movel([-0.046816, -1.563414, -2.421575, -0.727400, 1.570796, 1.523981],accel_mss,speed_ms,0,blend_radius_m)
    movel([-0.048058, -1.562711, -2.422269, -0.727409, 1.570796, 1.522738],accel_mss,speed_ms,0,blend_radius_m)
    movel([-0.049410, -1.562120, -2.422852, -0.727417, 1.570796, 1.521386],accel_mss,speed_ms,0,blend_radius_m)
    movel([-0.050857, -1.561642, -2.423323, -0.727424, 1.570796, 1.519939],accel_mss,speed_ms,0,blend_radius_m)
    movel([-0.052384, -1.561274, -2.423686, -0.727429, 1.570796, 1.518413],accel_mss,speed_ms,0,blend_radius_m)
    movel([-0.053976, -1.561017, -2.423938, -0.727433, 1.570796, 1.516821],accel_mss,speed_ms,0,blend_radius_m)
    movel([-0.055620, -1.560871, -2.424083, -0.727436, 1.570796, 1.515177],accel_mss,speed_ms,0,blend_radius_m)
    movel([-0.057299, -1.560831, -2.424122, -0.727436, 1.570796, 1.513497],accel_mss,speed_ms,0,blend_radius_m)
    movel([-0.058436, -1.560890, -2.424063, -0.727435, 1.570796, 1.512360],accel_mss,speed_ms,0,blend_radius_m)
    movel([-0.059341, -1.561045, -2.423911, -0.727433, 1.570796, 1.511456],accel_mss,speed_ms,0,blend_radius_m)
    movel([-0.060029, -1.561283, -2.423677, -0.727429, 1.570796, 1.510767],accel_mss,speed_ms,0,blend_radius_m)
    movel([-0.060522, -1.561594, -2.423370, -0.727425, 1.570796, 1.510275],accel_mss,speed_ms,0,blend_radius_m)
    movel([-0.060839, -1.561972, -2.422998, -0.727419, 1.570796, 1.509957],accel_mss,speed_ms,0,blend_radius_m)
    movel([-0.060998, -1.562406, -2.422570, -0.727413, 1.570796, 1.509798],accel_mss,speed_ms,0,blend_radius_m)
    movel([-0.061024, -1.562886, -2.422096, -0.727407, 1.570796, 1.509773],accel_mss,speed_ms,0,blend_radius_m)
    movel([-0.060930, -1.563404, -2.421585, -0.727400, 1.570796, 1.509866],accel_mss,speed_ms,0,blend_radius_m)
    movel([-0.060476, -1.564519, -2.420482, -0.727388, 1.570796, 1.510321],accel_mss,speed_ms,0,blend_radius_m)
    movel([-0.058367, -1.567859, -2.417166, -0.727363, 1.570796, 1.512429],accel_mss,speed_ms,0,blend_radius_m)
    movel([-0.059813, -1.566992, -2.418029, -0.727368, 1.570796, 1.510983],accel_mss,speed_ms,0,blend_radius_m)
    movel([-0.062636, -1.565198, -2.419810, -0.727382, 1.570796, 1.508160],accel_mss,speed_ms,0,blend_radius_m)
    movel([-0.064238, -1.564514, -2.420487, -0.727388, 1.570796, 1.506559],accel_mss,speed_ms,0,blend_radius_m)
    movel([-0.066175, -1.563972, -2.421023, -0.727394, 1.570796, 1.504621],accel_mss,speed_ms,0,blend_radius_m)
    movel([-0.068188, -1.563525, -2.421465, -0.727399, 1.570796, 1.502609],accel_mss,speed_ms,0,blend_radius_m)
    movel([-0.072264, -1.562702, -2.422278, -0.727409, 1.570796, 1.498533],accel_mss,speed_ms,0,blend_radius_m)
    movel([-0.074241, -1.562223, -2.422750, -0.727416, 1.570796, 1.496555],accel_mss,speed_ms,0,blend_radius_m)
    movel([-0.076119, -1.561629, -2.423336, -0.727424, 1.570796, 1.494677],accel_mss,speed_ms,0,blend_radius_m)
    movel([-0.077854, -1.560870, -2.424083, -0.727436, 1.570796, 1.492942],accel_mss,speed_ms,0,blend_radius_m)
    movel([-0.079405, -1.559889, -2.425047, -0.727452, 1.570796, 1.491391],accel_mss,speed_ms,0,blend_radius_m)
    movel([-0.078004, -1.562788, -2.422193, -0.727408, 1.570796, 1.492793],accel_mss,speed_ms,0,blend_radius_m)
    movel([-0.077190, -1.564223, -2.420774, -0.727391, 1.570796, 1.493606],accel_mss,speed_ms,0,blend_radius_m)
    movel([-0.076252, -1.565437, -2.419572, -0.727379, 1.570796, 1.494544],accel_mss,speed_ms,0,blend_radius_m)
    movel([-0.077828, -1.564527, -2.420474, -0.727388, 1.570796, 1.492968],accel_mss,speed_ms,0,blend_radius_m)
    movel([-0.079555, -1.563782, -2.421211, -0.727396, 1.570796, 1.491241],accel_mss,speed_ms,0,blend_radius_m)
    movel([-0.083157, -1.562454, -2.422523, -0.727412, 1.570796, 1.487639],accel_mss,speed_ms,0,blend_radius_m)
    movel([-0.084295, -1.561925, -2.423044, -0.727420, 1.570796, 1.486502],accel_mss,speed_ms,0,blend_radius_m)
    movel([-0.085304, -1.561305, -2.423655, -0.727429, 1.570796, 1.485493],accel_mss,speed_ms,0,blend_radius_m)
    movel([-0.087071, -1.559876, -2.425061, -0.727452, 1.570796, 1.483725],accel_mss,speed_ms,0,blend_radius_m)
    movel([-0.088743, -1.558350, -2.426558, -0.727481, 1.570796, 1.482053],accel_mss,speed_ms,0,blend_radius_m)
    movel([-0.090604, -1.556919, -2.427959, -0.727512, 1.570796, 1.480192],accel_mss,speed_ms,0,blend_radius_m)
    movel([-0.091273, -1.556544, -2.428325, -0.727520, 1.570796, 1.479524],accel_mss,speed_ms,0,blend_radius_m)
    movel([-0.092029, -1.556274, -2.428589, -0.727526, 1.570796, 1.478767],accel_mss,speed_ms,0,blend_radius_m)
    movel([-0.092868, -1.556196, -2.428664, -0.727528, 1.570796, 1.477929],accel_mss,speed_ms,0,blend_radius_m)
    movel([-0.093312, -1.556253, -2.428609, -0.727527, 1.570796, 1.477485],accel_mss,speed_ms,0,blend_radius_m)
    movel([-0.093773, -1.556392, -2.428473, -0.727524, 1.570796, 1.477023],accel_mss,speed_ms,0,blend_radius_m)
    movel([-0.094268, -1.556630, -2.428241, -0.727518, 1.570796, 1.476529],accel_mss,speed_ms,0,blend_radius_m)
    movel([-0.094711, -1.556935, -2.427942, -0.727511, 1.570796, 1.476085],accel_mss,speed_ms,0,blend_radius_m)
    movel([-0.095469, -1.557702, -2.427192, -0.727495, 1.570796, 1.475328],accel_mss,speed_ms,0,blend_radius_m)
    movel([-0.096070, -1.558593, -2.426319, -0.727476, 1.570796, 1.474726],accel_mss,speed_ms,0,blend_radius_m)
    movel([-0.096540, -1.559509, -2.425421, -0.727459, 1.570796, 1.474256],accel_mss,speed_ms,0,blend_radius_m)
    movel([-0.097023, -1.558082, -2.426821, -0.727487, 1.570796, 1.473773],accel_mss,speed_ms,0,blend_radius_m)
    movel([-0.097641, -1.556752, -2.428121, -0.727515, 1.570796, 1.473155],accel_mss,speed_ms,0,blend_radius_m)
    movel([-0.099137, -1.554288, -2.430525, -0.727576, 1.570796, 1.471659],accel_mss,speed_ms,0,blend_radius_m)
    movel([-0.100733, -1.551892, -2.432852, -0.727644, 1.570796, 1.470064],accel_mss,speed_ms,0,blend_radius_m)
    movel([-0.102125, -1.549338, -2.435323, -0.727727, 1.570796, 1.468671],accel_mss,speed_ms,0,blend_radius_m)
    movel([-0.102491, -1.548250, -2.436373, -0.727766, 1.570796, 1.468306],accel_mss,speed_ms,0,blend_radius_m)
    movel([-0.102692, -1.547057, -2.437521, -0.727811, 1.570796, 1.468104],accel_mss,speed_ms,0,blend_radius_m)
    movel([-0.102755, -1.545783, -2.438746, -0.727861, 1.570796, 1.468042],accel_mss,speed_ms,0,blend_radius_m)
    movel([-0.102703, -1.544455, -2.440019, -0.727916, 1.570796, 1.468094],accel_mss,speed_ms,0,blend_radius_m)
    movel([-0.102341, -1.541729, -2.442622, -0.728037, 1.570796, 1.468456],accel_mss,speed_ms,0,blend_radius_m)
    movel([-0.101797, -1.539085, -2.445137, -0.728167, 1.570796, 1.468999],accel_mss,speed_ms,0,blend_radius_m)
    speed_ms = 0.005
    movel([-0.101797, -1.531540, -2.441797, -0.739052, 1.570796, 1.468999],accel_mss,speed_ms,0,blend_radius_m)
    speed_ms = 0.040
    # Splitting Linear movement in 2 (instruction 806: MoveL 765)
    movel([-0.083040, -1.496373, -2.473790, -0.742226, 1.570796, 1.487756],accel_mss,speed_ms,0,blend_radius_m)
    movel([-0.062711, -1.459410, -2.505329, -0.747649, 1.570796, 1.508085],accel_mss,speed_ms,0,blend_radius_m)
    speed_ms = 0.005
    movel([-0.062711, -1.467532, -2.508951, -0.735906, 1.570796, 1.508085],accel_mss,speed_ms,0,blend_radius_m)
    speed_ms = 0.025
    movel([-0.063837, -1.468399, -2.508227, -0.735764, 1.570796, 1.506960],accel_mss,speed_ms,0,blend_radius_m)
    movel([-0.063923, -1.468577, -2.508077, -0.735735, 1.570796, 1.506874],accel_mss,speed_ms,0,blend_radius_m)
    movel([-0.063841, -1.468838, -2.507859, -0.735692, 1.570796, 1.506955],accel_mss,speed_ms,0,blend_radius_m)
    movel([-0.063219, -1.469593, -2.507226, -0.735570, 1.570796, 1.507577],accel_mss,speed_ms,0,blend_radius_m)
    movel([-0.060441, -1.471875, -2.505309, -0.735205, 1.570796, 1.510355],accel_mss,speed_ms,0,blend_radius_m)
    movel([-0.056183, -1.474894, -2.502759, -0.734736, 1.570796, 1.514613],accel_mss,speed_ms,0,blend_radius_m)
    movel([-0.051114, -1.478295, -2.499870, -0.734224, 1.570796, 1.519682],accel_mss,speed_ms,0,blend_radius_m)
    movel([-0.041146, -1.484794, -2.494299, -0.733297, 1.570796, 1.529651],accel_mss,speed_ms,0,blend_radius_m)
    movel([-0.035496, -1.488354, -2.491218, -0.732817, 1.570796, 1.535301],accel_mss,speed_ms,0,blend_radius_m)
    movel([-0.034943, -1.488610, -2.490996, -0.732783, 1.570796, 1.535853],accel_mss,speed_ms,0,blend_radius_m)
    movel([-0.034315, -1.488765, -2.490861, -0.732763, 1.570796, 1.536482],accel_mss,speed_ms,0,blend_radius_m)
    movel([-0.033650, -1.488731, -2.490891, -0.732767, 1.570796, 1.537147],accel_mss,speed_ms,0,blend_radius_m)
    movel([-0.033313, -1.488618, -2.490989, -0.732782, 1.570796, 1.537483],accel_mss,speed_ms,0,blend_radius_m)
    movel([-0.032983, -1.488424, -2.491157, -0.732807, 1.570796, 1.537814],accel_mss,speed_ms,0,blend_radius_m)
    movel([-0.032497, -1.487936, -2.491581, -0.732872, 1.570796, 1.538299],accel_mss,speed_ms,0,blend_radius_m)
    movel([-0.032145, -1.487377, -2.492066, -0.732946, 1.570796, 1.538651],accel_mss,speed_ms,0,blend_radius_m)
    movel([-0.030514, -1.484185, -2.494823, -0.733381, 1.570796, 1.540282],accel_mss,speed_ms,0,blend_radius_m)
    movel([-0.029155, -1.480964, -2.497589, -0.733835, 1.570796, 1.541641],accel_mss,speed_ms,0,blend_radius_m)
    movel([-0.028056, -1.477733, -2.500349, -0.734307, 1.570796, 1.542740],accel_mss,speed_ms,0,blend_radius_m)
    movel([-0.027194, -1.474507, -2.503087, -0.734795, 1.570796, 1.543603],accel_mss,speed_ms,0,blend_radius_m)
    movel([-0.026554, -1.471302, -2.505791, -0.735296, 1.570796, 1.544242],accel_mss,speed_ms,0,blend_radius_m)
    movel([-0.026117, -1.468135, -2.508447, -0.735807, 1.570796, 1.544679],accel_mss,speed_ms,0,blend_radius_m)
    movel([-0.025866, -1.465023, -2.511042, -0.736324, 1.570796, 1.544931],accel_mss,speed_ms,0,blend_radius_m)
    movel([-0.025780, -1.461986, -2.513560, -0.736843, 1.570796, 1.545016],accel_mss,speed_ms,0,blend_radius_m)
    movel([-0.025847, -1.460637, -2.514674, -0.737078, 1.570796, 1.544950],accel_mss,speed_ms,0,blend_radius_m)
    movel([-0.026050, -1.459421, -2.515675, -0.737292, 1.570796, 1.544746],accel_mss,speed_ms,0,blend_radius_m)
    movel([-0.026390, -1.458337, -2.516566, -0.737486, 1.570796, 1.544407],accel_mss,speed_ms,0,blend_radius_m)
    movel([-0.026856, -1.457380, -2.517351, -0.737657, 1.570796, 1.543941],accel_mss,speed_ms,0,blend_radius_m)
    movel([-0.027447, -1.456551, -2.518030, -0.737808, 1.570796, 1.543349],accel_mss,speed_ms,0,blend_radius_m)
    movel([-0.028158, -1.455848, -2.518605, -0.737936, 1.570796, 1.542638],accel_mss,speed_ms,0,blend_radius_m)
    movel([-0.028984, -1.455264, -2.519082, -0.738043, 1.570796, 1.541812],accel_mss,speed_ms,0,blend_radius_m)
    movel([-0.029921, -1.454799, -2.519462, -0.738128, 1.570796, 1.540875],accel_mss,speed_ms,0,blend_radius_m)
    movel([-0.030963, -1.454450, -2.519746, -0.738193, 1.570796, 1.539834],accel_mss,speed_ms,0,blend_radius_m)
    movel([-0.032104, -1.454214, -2.519938, -0.738236, 1.570796, 1.538692],accel_mss,speed_ms,0,blend_radius_m)
    movel([-0.033343, -1.454088, -2.520041, -0.738260, 1.570796, 1.537453],accel_mss,speed_ms,0,blend_radius_m)
    movel([-0.034670, -1.454070, -2.520056, -0.738263, 1.570796, 1.536126],accel_mss,speed_ms,0,blend_radius_m)
    movel([-0.037577, -1.454345, -2.519832, -0.738212, 1.570796, 1.533220],accel_mss,speed_ms,0,blend_radius_m)
    movel([-0.040780, -1.455010, -2.519289, -0.738089, 1.570796, 1.530016],accel_mss,speed_ms,0,blend_radius_m)
    movel([-0.043678, -1.455908, -2.518556, -0.737925, 1.570796, 1.527118],accel_mss,speed_ms,0,blend_radius_m)
    movel([-0.046535, -1.457075, -2.517601, -0.737713, 1.570796, 1.524261],accel_mss,speed_ms,0,blend_radius_m)
    movel([-0.049352, -1.458477, -2.516452, -0.737461, 1.570796, 1.521445],accel_mss,speed_ms,0,blend_radius_m)
    movel([-0.052124, -1.460068, -2.515143, -0.737178, 1.570796, 1.518673],accel_mss,speed_ms,0,blend_radius_m)
    movel([-0.054845, -1.461809, -2.513706, -0.736874, 1.570796, 1.515951],accel_mss,speed_ms,0,blend_radius_m)
    movel([-0.057519, -1.463659, -2.512174, -0.736555, 1.570796, 1.513277],accel_mss,speed_ms,0,blend_radius_m)
    movel([-0.062711, -1.467532, -2.508951, -0.735906, 1.570796, 1.508085],accel_mss,speed_ms,0,blend_radius_m)
    movel([-0.063837, -1.468399, -2.508227, -0.735764, 1.570796, 1.506960],accel_mss,speed_ms,0,blend_radius_m)
    movel([-0.063923, -1.468577, -2.508077, -0.735735, 1.570796, 1.506874],accel_mss,speed_ms,0,blend_radius_m)
    movel([-0.063841, -1.468838, -2.507859, -0.735692, 1.570796, 1.506955],accel_mss,speed_ms,0,blend_radius_m)
    movel([-0.063645, -1.469078, -2.507658, -0.735653, 1.570796, 1.507152],accel_mss,speed_ms,0,blend_radius_m)
    speed_ms = 0.005
    movel([-0.063645, -1.460968, -2.504043, -0.747378, 1.570796, 1.507152],accel_mss,speed_ms,0,blend_radius_m)
    speed_ms = 0.040
    movel([-0.072174, -1.446258, -2.516044, -0.750087, 1.570796, 1.498622],accel_mss,speed_ms,0,blend_radius_m)
    speed_ms = 0.005
    movel([-0.072174, -1.454482, -2.519720, -0.738187, 1.570796, 1.498622],accel_mss,speed_ms,0,blend_radius_m)
    speed_ms = 0.025
    movel([-0.072243, -1.453237, -2.520734, -0.738418, 1.570796, 1.498554],accel_mss,speed_ms,0,blend_radius_m)
    movel([-0.072544, -1.452088, -2.521667, -0.738634, 1.570796, 1.498253],accel_mss,speed_ms,0,blend_radius_m)
    movel([-0.073071, -1.451063, -2.522498, -0.738828, 1.570796, 1.497725],accel_mss,speed_ms,0,blend_radius_m)
    movel([-0.073812, -1.450185, -2.523208, -0.738996, 1.570796, 1.496985],accel_mss,speed_ms,0,blend_radius_m)
    movel([-0.076104, -1.448426, -2.524628, -0.739335, 1.570796, 1.494692],accel_mss,speed_ms,0,blend_radius_m)
    movel([-0.076657, -1.447844, -2.525096, -0.739448, 1.570796, 1.494140],accel_mss,speed_ms,0,blend_radius_m)
    movel([-0.077038, -1.447218, -2.525600, -0.739571, 1.570796, 1.493758],accel_mss,speed_ms,0,blend_radius_m)
    movel([-0.077170, -1.446555, -2.526133, -0.739701, 1.570796, 1.493626],accel_mss,speed_ms,0,blend_radius_m)
    movel([-0.076970, -1.445860, -2.526690, -0.739838, 1.570796, 1.493826],accel_mss,speed_ms,0,blend_radius_m)
    movel([-0.076391, -1.445103, -2.527297, -0.739989, 1.570796, 1.494405],accel_mss,speed_ms,0,blend_radius_m)
    movel([-0.075691, -1.444616, -2.527687, -0.740086, 1.570796, 1.495105],accel_mss,speed_ms,0,blend_radius_m)
    movel([-0.074908, -1.444355, -2.527895, -0.740138, 1.570796, 1.495888],accel_mss,speed_ms,0,blend_radius_m)
    movel([-0.074087, -1.444277, -2.527958, -0.740154, 1.570796, 1.496710],accel_mss,speed_ms,0,blend_radius_m)
    movel([-0.072504, -1.444494, -2.527784, -0.740111, 1.570796, 1.498293],accel_mss,speed_ms,0,blend_radius_m)
    movel([-0.071273, -1.444919, -2.527445, -0.740026, 1.570796, 1.499523],accel_mss,speed_ms,0,blend_radius_m)
    movel([-0.071721, -1.443489, -2.528587, -0.740313, 1.570796, 1.499075],accel_mss,speed_ms,0,blend_radius_m)
    movel([-0.072443, -1.442254, -2.529572, -0.740563, 1.570796, 1.498354],accel_mss,speed_ms,0,blend_radius_m)
    movel([-0.074382, -1.440116, -2.531271, -0.741002, 1.570796, 1.496414],accel_mss,speed_ms,0,blend_radius_m)
    movel([-0.076427, -1.437995, -2.532949, -0.741445, 1.570796, 1.494369],accel_mss,speed_ms,0,blend_radius_m)
    movel([-0.077282, -1.436778, -2.533909, -0.741702, 1.570796, 1.493514],accel_mss,speed_ms,0,blend_radius_m)
    movel([-0.077910, -1.435370, -2.535018, -0.742002, 1.570796, 1.492887],accel_mss,speed_ms,0,blend_radius_m)
    movel([-0.078155, -1.434398, -2.535780, -0.742211, 1.570796, 1.492641],accel_mss,speed_ms,0,blend_radius_m)
    movel([-0.078235, -1.433559, -2.536438, -0.742392, 1.570796, 1.492561],accel_mss,speed_ms,0,blend_radius_m)
    movel([-0.078168, -1.432849, -2.536994, -0.742547, 1.570796, 1.492628],accel_mss,speed_ms,0,blend_radius_m)
    movel([-0.077968, -1.432265, -2.537450, -0.742674, 1.570796, 1.492829],accel_mss,speed_ms,0,blend_radius_m)
    movel([-0.077656, -1.431807, -2.537808, -0.742775, 1.570796, 1.493140],accel_mss,speed_ms,0,blend_radius_m)
    movel([-0.077247, -1.431464, -2.538075, -0.742850, 1.570796, 1.493549],accel_mss,speed_ms,0,blend_radius_m)
    movel([-0.076762, -1.431238, -2.538251, -0.742900, 1.570796, 1.494034],accel_mss,speed_ms,0,blend_radius_m)
    movel([-0.076215, -1.431124, -2.538340, -0.742925, 1.570796, 1.494581],accel_mss,speed_ms,0,blend_radius_m)
    movel([-0.075625, -1.431117, -2.538345, -0.742926, 1.570796, 1.495171],accel_mss,speed_ms,0,blend_radius_m)
    movel([-0.075014, -1.431216, -2.538268, -0.742905, 1.570796, 1.495783],accel_mss,speed_ms,0,blend_radius_m)
    movel([-0.073786, -1.431708, -2.537885, -0.742796, 1.570796, 1.497010],accel_mss,speed_ms,0,blend_radius_m)
    movel([-0.072674, -1.432567, -2.537214, -0.742608, 1.570796, 1.498122],accel_mss,speed_ms,0,blend_radius_m)
    movel([-0.071818, -1.433760, -2.536280, -0.742348, 1.570796, 1.498978],accel_mss,speed_ms,0,blend_radius_m)
    movel([-0.071570, -1.432334, -2.537396, -0.742659, 1.570796, 1.499226],accel_mss,speed_ms,0,blend_radius_m)
    movel([-0.071523, -1.431037, -2.538408, -0.742944, 1.570796, 1.499273],accel_mss,speed_ms,0,blend_radius_m)
    movel([-0.071633, -1.429838, -2.539341, -0.743210, 1.570796, 1.499163],accel_mss,speed_ms,0,blend_radius_m)
    movel([-0.072441, -1.426473, -2.541948, -0.743968, 1.570796, 1.498355],accel_mss,speed_ms,0,blend_radius_m)
    movel([-0.072913, -1.424072, -2.543798, -0.744519, 1.570796, 1.497883],accel_mss,speed_ms,0,blend_radius_m)
    movel([-0.072968, -1.423023, -2.544604, -0.744762, 1.570796, 1.497829],accel_mss,speed_ms,0,blend_radius_m)
    movel([-0.072889, -1.422073, -2.545332, -0.744984, 1.570796, 1.497908],accel_mss,speed_ms,0,blend_radius_m)
    movel([-0.072695, -1.421230, -2.545977, -0.745182, 1.570796, 1.498101],accel_mss,speed_ms,0,blend_radius_m)
    movel([-0.072401, -1.420498, -2.546536, -0.745355, 1.570796, 1.498395],accel_mss,speed_ms,0,blend_radius_m)
    movel([-0.072027, -1.419881, -2.547006, -0.745502, 1.570796, 1.498770],accel_mss,speed_ms,0,blend_radius_m)
    movel([-0.071586, -1.419384, -2.547385, -0.745620, 1.570796, 1.499210],accel_mss,speed_ms,0,blend_radius_m)
    movel([-0.071096, -1.419012, -2.547668, -0.745709, 1.570796, 1.499700],accel_mss,speed_ms,0,blend_radius_m)
    movel([-0.070575, -1.418770, -2.547852, -0.745766, 1.570796, 1.500221],accel_mss,speed_ms,0,blend_radius_m)
    movel([-0.070039, -1.418663, -2.547934, -0.745792, 1.570796, 1.500757],accel_mss,speed_ms,0,blend_radius_m)
    movel([-0.069506, -1.418695, -2.547909, -0.745784, 1.570796, 1.501291],accel_mss,speed_ms,0,blend_radius_m)
    movel([-0.068990, -1.418869, -2.547777, -0.745743, 1.570796, 1.501806],accel_mss,speed_ms,0,blend_radius_m)
    movel([-0.068509, -1.419192, -2.547531, -0.745666, 1.570796, 1.502287],accel_mss,speed_ms,0,blend_radius_m)
